gfCNCPoint1[19237] = {X 519.7998, Y 70.9591, Z -2.1667, A 0.000, B 0.000, C 0.000 }
gfCNCPoint1[19238] = {X 517.4110, Y 70.8403, Z -2.1667, A 0.000, B 0.000, C 0.000 }
gfCNCPoint1[19239] = {X 515.0458, Y 70.4852, Z -2.1667, A 0.000, B 0.000, C 0.000 }
gfCNCPoint1[19240] = {X 512.7275, Y 69.8971, Z -2.1667, A 0.000, B 0.000, C 0.000 }
gfCNCPoint1[19241] = {X 510.4789, Y 69.0820, Z -2.1667, A 0.000, B 0.000, C 0.000 }
gfCNCPoint1[19242] = {X 509.6264, Y 68.7046, Z -2.1667, A 0.000, B 0.000, C 0.000 }
gfCNCPoint1[19243] = {X 508.7892, Y 68.2944, Z -2.1667, A 0.000, B 0.000, C 0.000 }
gfCNCPoint1[19244] = {X 507.1705, Y 68.6592, Z -2.1667, A 0.000, B 0.000, C 0.000 }
gfCNCPoint1[19245] = {X 505.5305, Y 68.9117, Z -2.1667, A 0.000, B 0.000, C 0.000 }
gfCNCPoint1[19246] = {X 504.1120, Y 69.0379, Z -2.1667, A 0.000, B 0.000, C 0.000 }
gfCNCPoint1[19247] = {X 502.6885, Y 69.0800, Z -2.1667, A 0.000, B 0.000, C 0.000 }
gfCNCPoint1[19248] = {X 502.0391, Y 69.0800, Z -2.1667, A 0.000, B 0.000, C 0.000 }
gfCNCPoint1[19249] = {X 501.1772, Y 71.1329, Z -2.1667, A 0.000, B 0.000, C 0.000 }
gfCNCPoint1[19250] = {X 500.1596, Y 73.1132, Z -2.1667, A 0.000, B 0.000, C 0.000 }
gfCNCPoint1[19251] = {X 500.1596, Y 73.6949, Z -2.1667, A 0.000, B 0.000, C 0.000 }
gfCNCPoint1[19252] = {X 507.6819, Y 73.6949, Z -2.1667, A 0.000, B 0.000, C 0.000 }
gfCNCPoint1[19253] = {X 507.6819, Y 76.0949, Z -2.1667, A 0.000, B 0.000, C 0.000 }
gfCNCPoint1[19254] = {X 576.0965, Y 76.0949, Z -2.1667, A 0.000, B 0.000, C 0.000 }
gfCNCPoint1[19255] = {X 576.0965, Y 72.8901, Z -2.1667, A 0.000, B 0.000, C 0.000 }
gfCNCPoint1[19256] = {X 575.7178, Y 72.8147, Z -2.1667, A 0.000, B 0.000, C 0.000 }
gfCNCPoint1[19257] = {X 575.3401, Y 72.7341, Z -2.1667, A 0.000, B 0.000, C 0.000 }
gfCNCPoint1[19258] = {X 573.3201, Y 73.1034, Z -2.1667, A 0.000, B 0.000, C 0.000 }
gfCNCPoint1[19259] = {X 571.2786, Y 73.3258, Z -2.1667, A 0.000, B 0.000, C 0.000 }
gfCNCPoint1[19260] = {X 569.2264, Y 73.4000, Z -2.1667, A 0.000, B 0.000, C 0.000 }
gfCNCPoint1[19261] = {X 562.4443, Y 73.4000, Z -2.1667, A 0.000, B 0.000, C 0.000 }
gfCNCPoint1[19262] = {X 560.3341, Y 73.3215, Z -2.1667, A 0.000, B 0.000, C 0.000 }
gfCNCPoint1[19263] = {X 558.2355, Y 73.0864, Z -2.1667, A 0.000, B 0.000, C 0.000 }
gfCNCPoint1[19264] = {X 556.1603, Y 72.6960, Z -2.1667, A 0.000, B 0.000, C 0.000 }
gfCNCPoint1[19265] = {X 554.1197, Y 72.1526, Z -2.1667, A 0.000, B 0.000, C 0.000 }
gfCNCPoint1[19266] = {X 552.1252, Y 71.4590, Z -2.1667, A 0.000, B 0.000, C 0.000 }
gfCNCPoint1[19267] = {X 549.9757, Y 70.5165, Z -2.1667, A 0.000, B 0.000, C 0.000 }
gfCNCPoint1[19268] = {X 547.9113, Y 69.3999, Z -2.1667, A 0.000, B 0.000, C 0.000 }
gfCNCPoint1[19269] = {X 545.9462, Y 68.1165, Z -2.1667, A 0.000, B 0.000, C 0.000 }
gfCNCPoint1[19270] = {X 544.0938, Y 66.6753, Z -2.1667, A 0.000, B 0.000, C 0.000 }
gfCNCPoint1[19271] = {X 543.8496, Y 66.6765, Z -2.1667, A 0.000, B 0.000, C 0.000 }
gfCNCPoint1[19272] = {X 543.6054, Y 66.6749, Z -2.1667, A 0.000, B 0.000, C 0.000 }
gfCNCPoint1[19273] = {X 529.2683, Y 66.6753, Z -2.1667, A 0.000, B 0.000, C 0.000 }
gfCNCPoint1[19274] = {X 527.1808, Y 67.4783, Z -2.1667, A 0.000, B 0.000, C 0.000 }
gfCNCPoint1[19275] = {X 525.0223, Y 68.0636, Z -2.1667, A 0.000, B 0.000, C 0.000 }
gfCNCPoint1[19276] = {X 522.8151, Y 68.4251, Z -2.1667, A 0.000, B 0.000, C 0.000 }
gfCNCPoint1[19277] = {X 520.5826, Y 68.5589, Z -2.1667, A 0.000, B 0.000, C 0.000 }
gfCNCPoint1[19278] = {X 519.7998, Y 68.5591, Z -2.1667, A 0.000, B 0.000, C 0.000 }
gfCNCPoint1[19279] = {X 517.5593, Y 68.4430, Z -2.1667, A 0.000, B 0.000, C 0.000 }
gfCNCPoint1[19280] = {X 515.3429, Y 68.0961, Z -2.1667, A 0.000, B 0.000, C 0.000 }
gfCNCPoint1[19281] = {X 513.1742, Y 67.5219, Z -2.1667, A 0.000, B 0.000, C 0.000 }
gfCNCPoint1[19282] = {X 511.0764, Y 66.7267, Z -2.1667, A 0.000, B 0.000, C 0.000 }
gfCNCPoint1[19283] = {X 509.0720, Y 65.7189, Z -2.1667, A 0.000, B 0.000, C 0.000 }
gfCNCPoint1[19284] = {X 506.9797, Y 66.2511, Z -2.1667, A 0.000, B 0.000, C 0.000 }
gfCNCPoint1[19285] = {X 504.8448, Y 66.5725, Z -2.1667, A 0.000, B 0.000, C 0.000 }
gfCNCPoint1[19286] = {X 502.6885, Y 66.6800, Z -2.1667, A 0.000, B 0.000, C 0.000 }
gfCNCPoint1[19287] = {X 500.3217, Y 66.6800, Z -2.1667, A 0.000, B 0.000, C 0.000 }
gfCNCPoint1[19288] = {X 499.6229, Y 68.6759, Z -2.1667, A 0.000, B 0.000, C 0.000 }
gfCNCPoint1[19289] = {X 498.7670, Y 70.6096, Z -2.1667, A 0.000, B 0.000, C 0.000 }
gfCNCPoint1[19290] = {X 497.7596, Y 72.4689, Z -2.1667, A 0.000, B 0.000, C 0.000 }
gfCNCPoint1[19291] = {X 497.7596, Y 76.0949, Z -2.1667, A 0.000, B 0.000, C 0.000 }
gfCNCPoint1[19292] = {X 507.6819, Y 76.0949, Z -2.1667, A 0.000, B 0.000, C 0.000 }
gfCNCPoint1[19293] = {X 507.6819, Y 78.4949, Z -2.1667, A 0.000, B 0.000, C 0.000 }
gfCNCPoint1[19294] = {X 578.4965, Y 78.4949, Z -2.1667, A 0.000, B 0.000, C 0.000 }
gfCNCPoint1[19295] = {X 578.4965, Y 70.8313, Z -2.1667, A 0.000, B 0.000, C 0.000 }
gfCNCPoint1[19296] = {X 576.9097, Y 70.5998, Z -2.1667, A 0.000, B 0.000, C 0.000 }
gfCNCPoint1[19297] = {X 575.3401, Y 70.2710, Z -2.1667, A 0.000, B 0.000, C 0.000 }
gfCNCPoint1[19298] = {X 573.3236, Y 70.6751, Z -2.1667, A 0.000, B 0.000, C 0.000 }
gfCNCPoint1[19299] = {X 571.2815, Y 70.9187, Z -2.1667, A 0.000, B 0.000, C 0.000 }
gfCNCPoint1[19300] = {X 569.2264, Y 71.0000, Z -2.1667, A 0.000, B 0.000, C 0.000 }
gfCNCPoint1[19301] = {X 562.4443, Y 71.0000, Z -2.1667, A 0.000, B 0.000, C 0.000 }
gfCNCPoint1[19302] = {X 560.0511, Y 70.8896, Z -2.1667, A 0.000, B 0.000, C 0.000 }
gfCNCPoint1[19303] = {X 557.6782, Y 70.5594, Z -2.1667, A 0.000, B 0.000, C 0.000 }
gfCNCPoint1[19304] = {X 555.3457, Y 70.0122, Z -2.1667, A 0.000, B 0.000, C 0.000 }
gfCNCPoint1[19305] = {X 553.0736, Y 69.2526, Z -2.1667, A 0.000, B 0.000, C 0.000 }
gfCNCPoint1[19306] = {X 550.8810, Y 68.2871, Z -2.1667, A 0.000, B 0.000, C 0.000 }
gfCNCPoint1[19307] = {X 548.7866, Y 67.1239, Z -2.1667, A 0.000, B 0.000, C 0.000 }
gfCNCPoint1[19308] = {X 546.8081, Y 65.7728, Z -2.1667, A 0.000, B 0.000, C 0.000 }
gfCNCPoint1[19309] = {X 544.9624, Y 64.2454, Z -2.1667, A 0.000, B 0.000, C 0.000 }
gfCNCPoint1[19310] = {X 544.2916, Y 64.2718, Z -2.1667, A 0.000, B 0.000, C 0.000 }
gfCNCPoint1[19311] = {X 543.6203, Y 64.2749, Z -2.1667, A 0.000, B 0.000, C 0.000 }
gfCNCPoint1[19312] = {X 528.7431, Y 64.2753, Z -2.1667, A 0.000, B 0.000, C 0.000 }
gfCNCPoint1[19313] = {X 526.7893, Y 65.0775, Z -2.1667, A 0.000, B 0.000, C 0.000 }
gfCNCPoint1[19314] = {X 524.7600, Y 65.6630, Z -2.1667, A 0.000, B 0.000, C 0.000 }
gfCNCPoint1[19315] = {X 522.6791, Y 66.0249, Z -2.1667, A 0.000, B 0.000, C 0.000 }
gfCNCPoint1[19316] = {X 520.5713, Y 66.1589, Z -2.1667, A 0.000, B 0.000, C 0.000 }
gfCNCPoint1[19317] = {X 519.7998, Y 66.1591, Z -2.1667, A 0.000, B 0.000, C 0.000 }
gfCNCPoint1[19318] = {X 517.9641, Y 66.0715, Z -2.1667, A 0.000, B 0.000, C 0.000 }
gfCNCPoint1[19319] = {X 516.1450, Y 65.8096, Z -2.1667, A 0.000, B 0.000, C 0.000 }
gfCNCPoint1[19320] = {X 514.3592, Y 65.3756, Z -2.1667, A 0.000, B 0.000, C 0.000 }
gfCNCPoint1[19321] = {X 512.6228, Y 64.7735, Z -2.1667, A 0.000, B 0.000, C 0.000 }
gfCNCPoint1[19322] = {X 510.9516, Y 64.0089, Z -2.1667, A 0.000, B 0.000, C 0.000 }
gfCNCPoint1[19323] = {X 509.3609, Y 63.0886, Z -2.1667, A 0.000, B 0.000, C 0.000 }
gfCNCPoint1[19324] = {X 507.7389, Y 63.6068, Z -2.1667, A 0.000, B 0.000, C 0.000 }
gfCNCPoint1[19325] = {X 506.0774, Y 63.9798, Z -2.1667, A 0.000, B 0.000, C 0.000 }
gfCNCPoint1[19326] = {X 504.3896, Y 64.2048, Z -2.1667, A 0.000, B 0.000, C 0.000 }
gfCNCPoint1[19327] = {X 502.6885, Y 64.2800, Z -2.1667, A 0.000, B 0.000, C 0.000 }
gfCNCPoint1[19328] = {X 498.4791, Y 64.2800, Z -2.1667, A 0.000, B 0.000, C 0.000 }
gfCNCPoint1[19329] = {X 497.9415, Y 66.2507, Z -2.1667, A 0.000, B 0.000, C 0.000 }
gfCNCPoint1[19330] = {X 497.2388, Y 68.1688, Z -2.1667, A 0.000, B 0.000, C 0.000 }
gfCNCPoint1[19331] = {X 496.3761, Y 70.0204, Z -2.1667, A 0.000, B 0.000, C 0.000 }
gfCNCPoint1[19332] = {X 495.3596, Y 71.7923, Z -2.1667, A 0.000, B 0.000, C 0.000 }
gfCNCPoint1[19333] = {X 495.3597, Y 78.4949, Z -2.1667, A 0.000, B 0.000, C 0.000 }
gfCNCPoint1[19334] = {X 507.6819, Y 78.4949, Z -2.1667, A 0.000, B 0.000, C 0.000 }
gfCNCPoint1[19335] = {X 507.6819, Y 80.8949, Z -2.1667, A 0.000, B 0.000, C 0.000 }
gfCNCPoint1[19336] = {X 580.8965, Y 80.8949, Z -2.1667, A 0.000, B 0.000, C 0.000 }
gfCNCPoint1[19337] = {X 580.8965, Y 68.5934, Z -2.1667, A 0.000, B 0.000, C 0.000 }
gfCNCPoint1[19338] = {X 579.0251, Y 68.4747, Z -2.1667, A 0.000, B 0.000, C 0.000 }
gfCNCPoint1[19339] = {X 577.1691, Y 68.2078, Z -2.1667, A 0.000, B 0.000, C 0.000 }
gfCNCPoint1[19340] = {X 575.3401, Y 67.7943, Z -2.1667, A 0.000, B 0.000, C 0.000 }
gfCNCPoint1[19341] = {X 573.3283, Y 68.2408, Z -2.1667, A 0.000, B 0.000, C 0.000 }
gfCNCPoint1[19342] = {X 571.2852, Y 68.5100, Z -2.1667, A 0.000, B 0.000, C 0.000 }
gfCNCPoint1[19343] = {X 569.2264, Y 68.6000, Z -2.1667, A 0.000, B 0.000, C 0.000 }
gfCNCPoint1[19344] = {X 562.4443, Y 68.6000, Z -2.1667, A 0.000, B 0.000, C 0.000 }
gfCNCPoint1[19345] = {X 560.1442, Y 68.4876, Z -2.1667, A 0.000, B 0.000, C 0.000 }
gfCNCPoint1[19346] = {X 557.8659, Y 68.1516, Z -2.1667, A 0.000, B 0.000, C 0.000 }
gfCNCPoint1[19347] = {X 555.6313, Y 67.5952, Z -2.1667, A 0.000, B 0.000, C 0.000 }
gfCNCPoint1[19348] = {X 553.4615, Y 66.8236, Z -2.1667, A 0.000, B 0.000, C 0.000 }
gfCNCPoint1[19349] = {X 551.3773, Y 65.8442, Z -2.1667, A 0.000, B 0.000, C 0.000 }
gfCNCPoint1[19350] = {X 549.3984, Y 64.6664, Z -2.1667, A 0.000, B 0.000, C 0.000 }
gfCNCPoint1[19351] = {X 547.5438, Y 63.3012, Z -2.1667, A 0.000, B 0.000, C 0.000 }
gfCNCPoint1[19352] = {X 545.8311, Y 61.7619, Z -2.1667, A 0.000, B 0.000, C 0.000 }
gfCNCPoint1[19353] = {X 544.7354, Y 61.8541, Z -2.1667, A 0.000, B 0.000, C 0.000 }
gfCNCPoint1[19354] = {X 543.6361, Y 61.8749, Z -2.1667, A 0.000, B 0.000, C 0.000 }
gfCNCPoint1[19355] = {X 528.1826, Y 61.8754, Z -2.1667, A 0.000, B 0.000, C 0.000 }
gfCNCPoint1[19356] = {X 526.3697, Y 62.6774, Z -2.1667, A 0.000, B 0.000, C 0.000 }
gfCNCPoint1[19357] = {X 524.4760, Y 63.2635, Z -2.1667, A 0.000, B 0.000, C 0.000 }
gfCNCPoint1[19358] = {X 522.5270, Y 63.6257, Z -2.1667, A 0.000, B 0.000, C 0.000 }
gfCNCPoint1[19359] = {X 520.5492, Y 63.7590, Z -2.1667, A 0.000, B 0.000, C 0.000 }
gfCNCPoint1[19360] = {X 519.7998, Y 63.7591, Z -2.1667, A 0.000, B 0.000, C 0.000 }
gfCNCPoint1[19361] = {X 517.9902, Y 63.6618, Z -2.1667, A 0.000, B 0.000, C 0.000 }
gfCNCPoint1[19362] = {X 516.2015, Y 63.3711, Z -2.1667, A 0.000, B 0.000, C 0.000 }
gfCNCPoint1[19363] = {X 514.4543, Y 62.8904, Z -2.1667, A 0.000, B 0.000, C 0.000 }
gfCNCPoint1[19364] = {X 512.7687, Y 62.2251, Z -2.1667, A 0.000, B 0.000, C 0.000 }
gfCNCPoint1[19365] = {X 511.1641, Y 61.3829, Z -2.1667, A 0.000, B 0.000, C 0.000 }
gfCNCPoint1[19366] = {X 509.6590, Y 60.3735, Z -2.1667, A 0.000, B 0.000, C 0.000 }
gfCNCPoint1[19367] = {X 507.9866, Y 61.0270, Z -2.1667, A 0.000, B 0.000, C 0.000 }
gfCNCPoint1[19368] = {X 506.2542, Y 61.4991, Z -2.1667, A 0.000, B 0.000, C 0.000 }
gfCNCPoint1[19369] = {X 504.4815, Y 61.7845, Z -2.1667, A 0.000, B 0.000, C 0.000 }
gfCNCPoint1[19370] = {X 502.6885, Y 61.8800, Z -2.1667, A 0.000, B 0.000, C 0.000 }
gfCNCPoint1[19371] = {X 496.4789, Y 61.8800, Z -2.1667, A 0.000, B 0.000, C 0.000 }
gfCNCPoint1[19372] = {X 496.1191, Y 63.8335, Z -2.1667, A 0.000, B 0.000, C 0.000 }
gfCNCPoint1[19373] = {X 495.5821, Y 65.7458, Z -2.1667, A 0.000, B 0.000, C 0.000 }
gfCNCPoint1[19374] = {X 494.8723, Y 67.6009, Z -2.1667, A 0.000, B 0.000, C 0.000 }
gfCNCPoint1[19375] = {X 493.9957, Y 69.3833, Z -2.1667, A 0.000, B 0.000, C 0.000 }
gfCNCPoint1[19376] = {X 492.9596, Y 71.0780, Z -2.1667, A 0.000, B 0.000, C 0.000 }
gfCNCPoint1[19377] = {X 492.9597, Y 80.8949, Z -2.1667, A 0.000, B 0.000, C 0.000 }
gfCNCPoint1[19378] = {X 507.6819, Y 80.8949, Z -2.1667, A 0.000, B 0.000, C 0.000 }
gfCNCPoint1[19379] = {X 507.6819, Y 83.2949, Z -2.1667, A 0.000, B 0.000, C 0.000 }
gfCNCPoint1[19380] = {X 583.2965, Y 83.2949, Z -2.1667, A 0.000, B 0.000, C 0.000 }
gfCNCPoint1[19381] = {X 583.2965, Y 66.1198, Z -2.1667, A 0.000, B 0.000, C 0.000 }
gfCNCPoint1[19382] = {X 581.2871, Y 66.1993, Z -2.1667, A 0.000, B 0.000, C 0.000 }
gfCNCPoint1[19383] = {X 579.2793, Y 66.0882, Z -2.1667, A 0.000, B 0.000, C 0.000 }
gfCNCPoint1[19384] = {X 577.2910, Y 65.7873, Z -2.1667, A 0.000, B 0.000, C 0.000 }
gfCNCPoint1[19385] = {X 575.3401, Y 65.2993, Z -2.1667, A 0.000, B 0.000, C 0.000 }
gfCNCPoint1[19386] = {X 573.3348, Y 65.7981, Z -2.1667, A 0.000, B 0.000, C 0.000 }
gfCNCPoint1[19387] = {X 571.2904, Y 66.0993, Z -2.1667, A 0.000, B 0.000, C 0.000 }
gfCNCPoint1[19388] = {X 569.2264, Y 66.2000, Z -2.1667, A 0.000, B 0.000, C 0.000 }
gfCNCPoint1[19389] = {X 562.4443, Y 66.2000, Z -2.1667, A 0.000, B 0.000, C 0.000 }
gfCNCPoint1[19390] = {X 560.2302, Y 66.0841, Z -2.1667, A 0.000, B 0.000, C 0.000 }
gfCNCPoint1[19391] = {X 558.0403, Y 65.7375, Z -2.1667, A 0.000, B 0.000, C 0.000 }
gfCNCPoint1[19392] = {X 555.8985, Y 65.1641, Z -2.1667, A 0.000, B 0.000, C 0.000 }
gfCNCPoint1[19393] = {X 553.8284, Y 64.3702, Z -2.1667, A 0.000, B 0.000, C 0.000 }
gfCNCPoint1[19394] = {X 551.8525, Y 63.3644, Z -2.1667, A 0.000, B 0.000, C 0.000 }
gfCNCPoint1[19395] = {X 549.9924, Y 62.1578, Z -2.1667, A 0.000, B 0.000, C 0.000 }
gfCNCPoint1[19396] = {X 548.2685, Y 60.7635, Z -2.1667, A 0.000, B 0.000, C 0.000 }
gfCNCPoint1[19397] = {X 546.6997, Y 59.1968, Z -2.1667, A 0.000, B 0.000, C 0.000 }
gfCNCPoint1[19398] = {X 545.1838, Y 59.4165, Z -2.1667, A 0.000, B 0.000, C 0.000 }
gfCNCPoint1[19399] = {X 543.6531, Y 59.4749, Z -2.1667, A 0.000, B 0.000, C 0.000 }
gfCNCPoint1[19400] = {X 527.5785, Y 59.4754, Z -2.1667, A 0.000, B 0.000, C 0.000 }
gfCNCPoint1[19401] = {X 525.9214, Y 60.2760, Z -2.1667, A 0.000, B 0.000, C 0.000 }
gfCNCPoint1[19402] = {X 524.1770, Y 60.8624, Z -2.1667, A 0.000, B 0.000, C 0.000 }
gfCNCPoint1[19403] = {X 522.3727, Y 61.2253, Z -2.1667, A 0.000, B 0.000, C 0.000 }
gfCNCPoint1[19404] = {X 520.5372, Y 61.3590, Z -2.1667, A 0.000, B 0.000, C 0.000 }
gfCNCPoint1[19405] = {X 519.7998, Y 61.3591, Z -2.1667, A 0.000, B 0.000, C 0.000 }
gfCNCPoint1[19406] = {X 518.0043, Y 61.2474, Z -2.1667, A 0.000, B 0.000, C 0.000 }
gfCNCPoint1[19407] = {X 516.2365, Y 60.9138, Z -2.1667, A 0.000, B 0.000, C 0.000 }
gfCNCPoint1[19408] = {X 514.5237, Y 60.3637, Z -2.1667, A 0.000, B 0.000, C 0.000 }
gfCNCPoint1[19409] = {X 512.8923, Y 59.6054, Z -2.1667, A 0.000, B 0.000, C 0.000 }
gfCNCPoint1[19410] = {X 511.3676, Y 58.6507, Z -2.1667, A 0.000, B 0.000, C 0.000 }
gfCNCPoint1[19411] = {X 509.9730, Y 57.5142, Z -2.1667, A 0.000, B 0.000, C 0.000 }
gfCNCPoint1[19412] = {X 508.6156, Y 58.2113, Z -2.1667, A 0.000, B 0.000, C 0.000 }
gfCNCPoint1[19413] = {X 507.1924, Y 58.7617, Z -2.1667, A 0.000, B 0.000, C 0.000 }
gfCNCPoint1[19414] = {X 505.7192, Y 59.1593, Z -2.1667, A 0.000, B 0.000, C 0.000 }
gfCNCPoint1[19415] = {X 504.2123, Y 59.3996, Z -2.1667, A 0.000, B 0.000, C 0.000 }
gfCNCPoint1[19416] = {X 502.6885, Y 59.4800, Z -2.1667, A 0.000, B 0.000, C 0.000 }
gfCNCPoint1[19417] = {X 496.2450, Y 59.4800, Z -2.1667, A 0.000, B 0.000, C 0.000 }
gfCNCPoint1[19418] = {X 495.2580, Y 59.4463, Z -2.1667, A 0.000, B 0.000, C 0.000 }
gfCNCPoint1[19419] = {X 494.2756, Y 59.3454, Z -2.1667, A 0.000, B 0.000, C 0.000 }
gfCNCPoint1[19420] = {X 494.1342, Y 61.3007, Z -2.1667, A 0.000, B 0.000, C 0.000 }
gfCNCPoint1[19421] = {X 493.7949, Y 63.2316, Z -2.1667, A 0.000, B 0.000, C 0.000 }
gfCNCPoint1[19422] = {X 493.2614, Y 65.1180, Z -2.1667, A 0.000, B 0.000, C 0.000 }
gfCNCPoint1[19423] = {X 492.5390, Y 66.9405, Z -2.1667, A 0.000, B 0.000, C 0.000 }
gfCNCPoint1[19424] = {X 491.6353, Y 68.6801, Z -2.1667, A 0.000, B 0.000, C 0.000 }
gfCNCPoint1[19425] = {X 490.5596, Y 70.3191, Z -2.1667, A 0.000, B 0.000, C 0.000 }
gfCNCPoint1[19426] = {X 490.5597, Y 83.2949, Z -2.1667, A 0.000, B 0.000, C 0.000 }
gfCNCPoint1[19427] = {X 507.6819, Y 83.2949, Z -2.1667, A 0.000, B 0.000, C 0.000 }
gfCNCPoint1[19428] = {X 507.6819, Y 85.6949, Z -2.1667, A 0.000, B 0.000, C 0.000 }
gfCNCPoint1[19429] = {X 585.6965, Y 85.6949, Z -2.1667, A 0.000, B 0.000, C 0.000 }
gfCNCPoint1[19430] = {X 585.6965, Y 63.3150, Z -2.1667, A 0.000, B 0.000, C 0.000 }
gfCNCPoint1[19431] = {X 584.3995, Y 63.5678, Z -2.1667, A 0.000, B 0.000, C 0.000 }
gfCNCPoint1[19432] = {X 583.0879, Y 63.7289, Z -2.1667, A 0.000, B 0.000, C 0.000 }
gfCNCPoint1[19433] = {X 581.1242, Y 63.7971, Z -2.1667, A 0.000, B 0.000, C 0.000 }
gfCNCPoint1[19434] = {X 579.1641, Y 63.6600, Z -2.1667, A 0.000, B 0.000, C 0.000 }
gfCNCPoint1[19435] = {X 577.2291, Y 63.3191, Z -2.1667, A 0.000, B 0.000, C 0.000 }
gfCNCPoint1[19436] = {X 575.3401, Y 62.7781, Z -2.1667, A 0.000, B 0.000, C 0.000 }
gfCNCPoint1[19437] = {X 573.3441, Y 63.3435, Z -2.1667, A 0.000, B 0.000, C 0.000 }
gfCNCPoint1[19438] = {X 571.2979, Y 63.6855, Z -2.1667, A 0.000, B 0.000, C 0.000 }
gfCNCPoint1[19439] = {X 569.2264, Y 63.8000, Z -2.1667, A 0.000, B 0.000, C 0.000 }
gfCNCPoint1[19440] = {X 562.4443, Y 63.8000, Z -2.1667, A 0.000, B 0.000, C 0.000 }
gfCNCPoint1[19441] = {X 560.5407, Y 63.7034, Z -2.1667, A 0.000, B 0.000, C 0.000 }
gfCNCPoint1[19442] = {X 558.6566, Y 63.4145, Z -2.1667, A 0.000, B 0.000, C 0.000 }
gfCNCPoint1[19443] = {X 556.8115, Y 62.9363, Z -2.1667, A 0.000, B 0.000, C 0.000 }
gfCNCPoint1[19444] = {X 555.0242, Y 62.2737, Z -2.1667, A 0.000, B 0.000, C 0.000 }
gfCNCPoint1[19445] = {X 553.3133, Y 61.4336, Z -2.1667, A 0.000, B 0.000, C 0.000 }
gfCNCPoint1[19446] = {X 551.6962, Y 60.4246, Z -2.1667, A 0.000, B 0.000, C 0.000 }
gfCNCPoint1[19447] = {X 550.1896, Y 59.2570, Z -2.1667, A 0.000, B 0.000, C 0.000 }
gfCNCPoint1[19448] = {X 548.8089, Y 57.9428, Z -2.1667, A 0.000, B 0.000, C 0.000 }
gfCNCPoint1[19449] = {X 547.5685, Y 56.4956, Z -2.1667, A 0.000, B 0.000, C 0.000 }
gfCNCPoint1[19450] = {X 546.2932, Y 56.8304, Z -2.1667, A 0.000, B 0.000, C 0.000 }
gfCNCPoint1[19451] = {X 544.9891, Y 57.0243, Z -2.1667, A 0.000, B 0.000, C 0.000 }
gfCNCPoint1[19452] = {X 543.6716, Y 57.0749, Z -2.1667, A 0.000, B 0.000, C 0.000 }
gfCNCPoint1[19453] = {X 526.9187, Y 57.0754, Z -2.1667, A 0.000, B 0.000, C 0.000 }
gfCNCPoint1[19454] = {X 525.4309, Y 57.8752, Z -2.1667, A 0.000, B 0.000, C 0.000 }
gfCNCPoint1[19455] = {X 523.8471, Y 58.4624, Z -2.1667, A 0.000, B 0.000, C 0.000 }
gfCNCPoint1[19456] = {X 522.1975, Y 58.8261, Z -2.1667, A 0.000, B 0.000, C 0.000 }
gfCNCPoint1[19457] = {X 520.5136, Y 58.9591, Z -2.1667, A 0.000, B 0.000, C 0.000 }
gfCNCPoint1[19458] = {X 519.7998, Y 58.9591, Z -2.1667, A 0.000, B 0.000, C 0.000 }
gfCNCPoint1[19459] = {X 518.2467, Y 58.8589, Z -2.1667, A 0.000, B 0.000, C 0.000 }
gfCNCPoint1[19460] = {X 516.7195, Y 58.5598, Z -2.1667, A 0.000, B 0.000, C 0.000 }
gfCNCPoint1[19461] = {X 515.2433, Y 58.0668, Z -2.1667, A 0.000, B 0.000, C 0.000 }
gfCNCPoint1[19462] = {X 513.8428, Y 57.3882, Z -2.1667, A 0.000, B 0.000, C 0.000 }
gfCNCPoint1[19463] = {X 512.5411, Y 56.5351, Z -2.1667, A 0.000, B 0.000, C 0.000 }
gfCNCPoint1[19464] = {X 511.3600, Y 55.5218, Z -2.1667, A 0.000, B 0.000, C 0.000 }
gfCNCPoint1[19465] = {X 510.3189, Y 54.3650, Z -2.1667, A 0.000, B 0.000, C 0.000 }
gfCNCPoint1[19466] = {X 508.9711, Y 55.3177, Z -2.1667, A 0.000, B 0.000, C 0.000 }
gfCNCPoint1[19467] = {X 507.5060, Y 56.0778, Z -2.1667, A 0.000, B 0.000, C 0.000 }
gfCNCPoint1[19468] = {X 505.9510, Y 56.6311, Z -2.1667, A 0.000, B 0.000, C 0.000 }
gfCNCPoint1[19469] = {X 504.3351, Y 56.9672, Z -2.1667, A 0.000, B 0.000, C 0.000 }
gfCNCPoint1[19470] = {X 502.6885, Y 57.0800, Z -2.1667, A 0.000, B 0.000, C 0.000 }
gfCNCPoint1[19471] = {X 496.2450, Y 57.0800, Z -2.1667, A 0.000, B 0.000, C 0.000 }
gfCNCPoint1[19472] = {X 495.4216, Y 57.0519, Z -2.1667, A 0.000, B 0.000, C 0.000 }
gfCNCPoint1[19473] = {X 494.6020, Y 56.9677, Z -2.1667, A 0.000, B 0.000, C 0.000 }
gfCNCPoint1[19474] = {X 493.1719, Y 56.6826, Z -2.1667, A 0.000, B 0.000, C 0.000 }
gfCNCPoint1[19475] = {X 491.7866, Y 56.2272, Z -2.1667, A 0.000, B 0.000, C 0.000 }
gfCNCPoint1[19476] = {X 491.8566, Y 57.1124, Z -2.1667, A 0.000, B 0.000, C 0.000 }
gfCNCPoint1[19477] = {X 491.8800, Y 58.0000, Z -2.1667, A 0.000, B 0.000, C 0.000 }
gfCNCPoint1[19478] = {X 491.8794, Y 59.0735, Z -2.1667, A 0.000, B 0.000, C 0.000 }
gfCNCPoint1[19479] = {X 491.8781, Y 59.1839, Z -2.1667, A 0.000, B 0.000, C 0.000 }
gfCNCPoint1[19480] = {X 491.8762, Y 59.2942, Z -2.1667, A 0.000, B 0.000, C 0.000 }
gfCNCPoint1[19481] = {X 491.7363, Y 61.1320, Z -2.1667, A 0.000, B 0.000, C 0.000 }
gfCNCPoint1[19482] = {X 491.3969, Y 62.9435, Z -2.1667, A 0.000, B 0.000, C 0.000 }
gfCNCPoint1[19483] = {X 490.8621, Y 64.7072, Z -2.1667, A 0.000, B 0.000, C 0.000 }
gfCNCPoint1[19484] = {X 490.1381, Y 66.4022, Z -2.1667, A 0.000, B 0.000, C 0.000 }
gfCNCPoint1[19485] = {X 489.2337, Y 68.0080, Z -2.1667, A 0.000, B 0.000, C 0.000 }
gfCNCPoint1[19486] = {X 488.1596, Y 69.5057, Z -2.1667, A 0.000, B 0.000, C 0.000 }
gfCNCPoint1[19487] = {X 488.1598, Y 85.6949, Z -2.1667, A 0.000, B 0.000, C 0.000 }
gfCNCPoint1[19488] = {X 507.6819, Y 85.6949, Z -2.1667, A 0.000, B 0.000, C 0.000 }
gfCNCPoint1[19489] = {X 507.6819, Y 88.0949, Z -2.1667, A 0.000, B 0.000, C 0.000 }
gfCNCPoint1[19490] = {X 588.0965, Y 88.0949, Z -2.1667, A 0.000, B 0.000, C 0.000 }
gfCNCPoint1[19491] = {X 588.0965, Y 60.4644, Z -2.1667, A 0.000, B 0.000, C 0.000 }
gfCNCPoint1[19492] = {X 587.7998, Y 60.3564, Z -2.1667, A 0.000, B 0.000, C 0.000 }
gfCNCPoint1[19493] = {X 587.5052, Y 60.2427, Z -2.1667, A 0.000, B 0.000, C 0.000 }
gfCNCPoint1[19494] = {X 586.3438, Y 60.6540, Z -2.1667, A 0.000, B 0.000, C 0.000 }
gfCNCPoint1[19495] = {X 585.1549, Y 60.9769, Z -2.1667, A 0.000, B 0.000, C 0.000 }
gfCNCPoint1[19496] = {X 583.5152, Y 61.2699, Z -2.1667, A 0.000, B 0.000, C 0.000 }
gfCNCPoint1[19497] = {X 581.8543, Y 61.3951, Z -2.1667, A 0.000, B 0.000, C 0.000 }
gfCNCPoint1[19498] = {X 580.1892, Y 61.3512, Z -2.1667, A 0.000, B 0.000, C 0.000 }
gfCNCPoint1[19499] = {X 578.5372, Y 61.1386, Z -2.1667, A 0.000, B 0.000, C 0.000 }
gfCNCPoint1[19500] = {X 576.9153, Y 60.7595, Z -2.1667, A 0.000, B 0.000, C 0.000 }
gfCNCPoint1[19501] = {X 575.3401, Y 60.2178, Z -2.1667, A 0.000, B 0.000, C 0.000 }
gfCNCPoint1[19502] = {X 573.8611, Y 60.7315, Z -2.1667, A 0.000, B 0.000, C 0.000 }
gfCNCPoint1[19503] = {X 572.3399, Y 61.1017, Z -2.1667, A 0.000, B 0.000, C 0.000 }
gfCNCPoint1[19504] = {X 570.7903, Y 61.3253, Z -2.1667, A 0.000, B 0.000, C 0.000 }
gfCNCPoint1[19505] = {X 569.2264, Y 61.4000, Z -2.1667, A 0.000, B 0.000, C 0.000 }
gfCNCPoint1[19506] = {X 562.4443, Y 61.4000, Z -2.1667, A 0.000, B 0.000, C 0.000 }
gfCNCPoint1[19507] = {X 560.5827, Y 61.2940, Z -2.1667, A 0.000, B 0.000, C 0.000 }
gfCNCPoint1[19508] = {X 558.7453, Y 60.9774, Z -2.1667, A 0.000, B 0.000, C 0.000 }
gfCNCPoint1[19509] = {X 556.9556, Y 60.4543, Z -2.1667, A 0.000, B 0.000, C 0.000 }
gfCNCPoint1[19510] = {X 555.2369, Y 59.7313, Z -2.1667, A 0.000, B 0.000, C 0.000 }
gfCNCPoint1[19511] = {X 553.6113, Y 58.8180, Z -2.1667, A 0.000, B 0.000, C 0.000 }
gfCNCPoint1[19512] = {X 552.0999, Y 57.7261, Z -2.1667, A 0.000, B 0.000, C 0.000 }
gfCNCPoint1[19513] = {X 550.7222, Y 56.4697, Z -2.1667, A 0.000, B 0.000, C 0.000 }
gfCNCPoint1[19514] = {X 549.4961, Y 55.0650, Z -2.1667, A 0.000, B 0.000, C 0.000 }
gfCNCPoint1[19515] = {X 548.4373, Y 53.5302, Z -2.1667, A 0.000, B 0.000, C 0.000 }
gfCNCPoint1[19516] = {X 547.3156, Y 54.0416, Z -2.1667, A 0.000, B 0.000, C 0.000 }
gfCNCPoint1[19517] = {X 546.1380, Y 54.4064, Z -2.1667, A 0.000, B 0.000, C 0.000 }
gfCNCPoint1[19518] = {X 544.9235, Y 54.6187, Z -2.1667, A 0.000, B 0.000, C 0.000 }
gfCNCPoint1[19519] = {X 543.6920, Y 54.6749, Z -2.1667, A 0.000, B 0.000, C 0.000 }
gfCNCPoint1[19520] = {X 526.1842, Y 54.6754, Z -2.1667, A 0.000, B 0.000, C 0.000 }
gfCNCPoint1[19521] = {X 524.8903, Y 55.4721, Z -2.1667, A 0.000, B 0.000, C 0.000 }
gfCNCPoint1[19522] = {X 523.4892, Y 56.0601, Z -2.1667, A 0.000, B 0.000, C 0.000 }
gfCNCPoint1[19523] = {X 522.0142, Y 56.4254, Z -2.1667, A 0.000, B 0.000, C 0.000 }
gfCNCPoint1[19524] = {X 520.5006, Y 56.5591, Z -2.1667, A 0.000, B 0.000, C 0.000 }
gfCNCPoint1[19525] = {X 519.7998, Y 56.5591, Z -2.1667, A 0.000, B 0.000, C 0.000 }
gfCNCPoint1[19526] = {X 518.3493, Y 56.4498, Z -2.1667, A 0.000, B 0.000, C 0.000 }
gfCNCPoint1[19527] = {X 516.9316, Y 56.1244, Z -2.1667, A 0.000, B 0.000, C 0.000 }
gfCNCPoint1[19528] = {X 515.5787, Y 55.5903, Z -2.1667, A 0.000, B 0.000, C 0.000 }
gfCNCPoint1[19529] = {X 514.3210, Y 54.8595, Z -2.1667, A 0.000, B 0.000, C 0.000 }
gfCNCPoint1[19530] = {X 513.1871, Y 53.9484, Z -2.1667, A 0.000, B 0.000, C 0.000 }
gfCNCPoint1[19531] = {X 512.2025, Y 52.8778, Z -2.1667, A 0.000, B 0.000, C 0.000 }
gfCNCPoint1[19532] = {X 511.3855, Y 51.6648, Z -2.1667, A 0.000, B 0.000, C 0.000 }
gfCNCPoint1[19533] = {X 510.7606, Y 50.3426, Z -2.1667, A 0.000, B 0.000, C 0.000 }
gfCNCPoint1[19534] = {X 509.8636, Y 51.4977, Z -2.1667, A 0.000, B 0.000, C 0.000 }
gfCNCPoint1[19535] = {X 508.8029, Y 52.5044, Z -2.1667, A 0.000, B 0.000, C 0.000 }
gfCNCPoint1[19536] = {X 507.7229, Y 53.2678, Z -2.1667, A 0.000, B 0.000, C 0.000 }
gfCNCPoint1[19537] = {X 506.5489, Y 53.8769, Z -2.1667, A 0.000, B 0.000, C 0.000 }
gfCNCPoint1[19538] = {X 505.3028, Y 54.3203, Z -2.1667, A 0.000, B 0.000, C 0.000 }
gfCNCPoint1[19539] = {X 504.0080, Y 54.5896, Z -2.1667, A 0.000, B 0.000, C 0.000 }
gfCNCPoint1[19540] = {X 502.6885, Y 54.6800, Z -2.1667, A 0.000, B 0.000, C 0.000 }
gfCNCPoint1[19541] = {X 496.2450, Y 54.6800, Z -2.1667, A 0.000, B 0.000, C 0.000 }
gfCNCPoint1[19542] = {X 495.0285, Y 54.6033, Z -2.1667, A 0.000, B 0.000, C 0.000 }
gfCNCPoint1[19543] = {X 493.8313, Y 54.3742, Z -2.1667, A 0.000, B 0.000, C 0.000 }
gfCNCPoint1[19544] = {X 492.6724, Y 53.9966, Z -2.1667, A 0.000, B 0.000, C 0.000 }
gfCNCPoint1[19545] = {X 491.4451, Y 53.4062, Z -2.1667, A 0.000, B 0.000, C 0.000 }
gfCNCPoint1[19546] = {X 490.3129, Y 52.6493, Z -2.1667, A 0.000, B 0.000, C 0.000 }
gfCNCPoint1[19547] = {X 489.2980, Y 51.7410, Z -2.1667, A 0.000, B 0.000, C 0.000 }
gfCNCPoint1[19548] = {X 488.8683, Y 52.1573, Z -2.1667, A 0.000, B 0.000, C 0.000 }
gfCNCPoint1[19549] = {X 488.4137, Y 52.5463, Z -2.1667, A 0.000, B 0.000, C 0.000 }
gfCNCPoint1[19550] = {X 488.8649, Y 53.8245, Z -2.1667, A 0.000, B 0.000, C 0.000 }
gfCNCPoint1[19551] = {X 489.1946, Y 55.1393, Z -2.1667, A 0.000, B 0.000, C 0.000 }
gfCNCPoint1[19552] = {X 489.3999, Y 56.4792, Z -2.1667, A 0.000, B 0.000, C 0.000 }
gfCNCPoint1[19553] = {X 489.4600, Y 57.2386, Z -2.1667, A 0.000, B 0.000, C 0.000 }
gfCNCPoint1[19554] = {X 489.4800, Y 58.0000, Z -2.1667, A 0.000, B 0.000, C 0.000 }
gfCNCPoint1[19555] = {X 489.4795, Y 59.0537, Z -2.1667, A 0.000, B 0.000, C 0.000 }
gfCNCPoint1[19556] = {X 489.3595, Y 60.7979, Z -2.1667, A 0.000, B 0.000, C 0.000 }
gfCNCPoint1[19557] = {X 489.0302, Y 62.5150, Z -2.1667, A 0.000, B 0.000, C 0.000 }
gfCNCPoint1[19558] = {X 488.4964, Y 64.1799, Z -2.1667, A 0.000, B 0.000, C 0.000 }
gfCNCPoint1[19559] = {X 487.7657, Y 65.7682, Z -2.1667, A 0.000, B 0.000, C 0.000 }
gfCNCPoint1[19560] = {X 486.8490, Y 67.2570, Z -2.1667, A 0.000, B 0.000, C 0.000 }
gfCNCPoint1[19561] = {X 485.7595, Y 68.6244, Z -2.1667, A 0.000, B 0.000, C 0.000 }
gfCNCPoint1[19562] = {X 485.7598, Y 87.3800, Z -2.1667, A 0.000, B 0.000, C 0.000 }
gfCNCPoint1[19563] = {X 486.0676, Y 87.7326, Z -2.1667, A 0.000, B 0.000, C 0.000 }
gfCNCPoint1[19564] = {X 486.3638, Y 88.0949, Z -2.1667, A 0.000, B 0.000, C 0.000 }
gfCNCPoint1[19565] = {X 507.6819, Y 88.0949, Z -2.1667, A 0.000, B 0.000, C 0.000 }
gfCNCPoint1[19566] = {X 507.6819, Y 90.4949, Z -2.1667, A 0.000, B 0.000, C 0.000 }
gfCNCPoint1[19567] = {X 590.4965, Y 90.4949, Z -2.1667, A 0.000, B 0.000, C 0.000 }
gfCNCPoint1[19568] = {X 590.4965, Y 58.6615, Z -2.1667, A 0.000, B 0.000, C 0.000 }
gfCNCPoint1[19569] = {X 588.9714, Y 58.2279, Z -2.1667, A 0.000, B 0.000, C 0.000 }
gfCNCPoint1[19570] = {X 587.5052, Y 57.6246, Z -2.1667, A 0.000, B 0.000, C 0.000 }
gfCNCPoint1[19571] = {X 585.8387, Y 58.2956, Z -2.1667, A 0.000, B 0.000, C 0.000 }
gfCNCPoint1[19572] = {X 584.0999, Y 58.7477, Z -2.1667, A 0.000, B 0.000, C 0.000 }
gfCNCPoint1[19573] = {X 582.3176, Y 58.9733, Z -2.1667, A 0.000, B 0.000, C 0.000 }
gfCNCPoint1[19574] = {X 580.5210, Y 58.9689, Z -2.1667, A 0.000, B 0.000, C 0.000 }
gfCNCPoint1[19575] = {X 578.7398, Y 58.7344, Z -2.1667, A 0.000, B 0.000, C 0.000 }
gfCNCPoint1[19576] = {X 577.0034, Y 58.2738, Z -2.1667, A 0.000, B 0.000, C 0.000 }
gfCNCPoint1[19577] = {X 575.3401, Y 57.5945, Z -2.1667, A 0.000, B 0.000, C 0.000 }
gfCNCPoint1[19578] = {X 573.8813, Y 58.2035, Z -2.1667, A 0.000, B 0.000, C 0.000 }
gfCNCPoint1[19579] = {X 572.3630, Y 58.6441, Z -2.1667, A 0.000, B 0.000, C 0.000 }
gfCNCPoint1[19580] = {X 570.8048, Y 58.9107, Z -2.1667, A 0.000, B 0.000, C 0.000 }
gfCNCPoint1[19581] = {X 569.2264, Y 59.0000, Z -2.1667, A 0.000, B 0.000, C 0.000 }
gfCNCPoint1[19582] = {X 562.4443, Y 59.0000, Z -2.1667, A 0.000, B 0.000, C 0.000 }
gfCNCPoint1[19583] = {X 560.6576, Y 58.8855, Z -2.1667, A 0.000, B 0.000, C 0.000 }
gfCNCPoint1[19584] = {X 558.9000, Y 58.5439, Z -2.1667, A 0.000, B 0.000, C 0.000 }
gfCNCPoint1[19585] = {X 557.2005, Y 57.9808, Z -2.1667, A 0.000, B 0.000, C 0.000 }
gfCNCPoint1[19586] = {X 555.5867, Y 57.2054, Z -2.1667, A 0.000, B 0.000, C 0.000 }
gfCNCPoint1[19587] = {X 554.0850, Y 56.2304, Z -2.1667, A 0.000, B 0.000, C 0.000 }
gfCNCPoint1[19588] = {X 552.7201, Y 55.0717, Z -2.1667, A 0.000, B 0.000, C 0.000 }
gfCNCPoint1[19589] = {X 551.5142, Y 53.7483, Z -2.1667, A 0.000, B 0.000, C 0.000 }
gfCNCPoint1[19590] = {X 550.4871, Y 52.2818, Z -2.1667, A 0.000, B 0.000, C 0.000 }
gfCNCPoint1[19591] = {X 549.8374, Y 51.0881, Z -2.1667, A 0.000, B 0.000, C 0.000 }
gfCNCPoint1[19592] = {X 549.3065, Y 49.8371, Z -2.1667, A 0.000, B 0.000, C 0.000 }
gfCNCPoint1[19593] = {X 548.3751, Y 50.7139, Z -2.1667, A 0.000, B 0.000, C 0.000 }
gfCNCPoint1[19594] = {X 547.3047, Y 51.4142, Z -2.1667, A 0.000, B 0.000, C 0.000 }
gfCNCPoint1[19595] = {X 546.1632, Y 51.9051, Z -2.1667, A 0.000, B 0.000, C 0.000 }
gfCNCPoint1[19596] = {X 544.9550, Y 52.1948, Z -2.1667, A 0.000, B 0.000, C 0.000 }
gfCNCPoint1[19597] = {X 543.7152, Y 52.2749, Z -2.1667, A 0.000, B 0.000, C 0.000 }
gfCNCPoint1[19598] = {X 525.3420, Y 52.2754, Z -2.1667, A 0.000, B 0.000, C 0.000 }
gfCNCPoint1[19599] = {X 524.2749, Y 53.0670, Z -2.1667, A 0.000, B 0.000, C 0.000 }
gfCNCPoint1[19600] = {X 523.0841, Y 53.6562, Z -2.1667, A 0.000, B 0.000, C 0.000 }
gfCNCPoint1[19601] = {X 521.8075, Y 54.0241, Z -2.1667, A 0.000, B 0.000, C 0.000 }
gfCNCPoint1[19602] = {X 520.4857, Y 54.1591, Z -2.1667, A 0.000, B 0.000, C 0.000 }
gfCNCPoint1[19603] = {X 519.7998, Y 54.1591, Z -2.1667, A 0.000, B 0.000, C 0.000 }
gfCNCPoint1[19604] = {X 518.5529, Y 54.0515, Z -2.1667, A 0.000, B 0.000, C 0.000 }
gfCNCPoint1[19605] = {X 517.3428, Y 53.7320, Z -2.1667, A 0.000, B 0.000, C 0.000 }
gfCNCPoint1[19606] = {X 516.2054, Y 53.2099, Z -2.1667, A 0.000, B 0.000, C 0.000 }
gfCNCPoint1[19607] = {X 515.1742, Y 52.5007, Z -2.1667, A 0.000, B 0.000, C 0.000 }
gfCNCPoint1[19608] = {X 514.2797, Y 51.6254, Z -2.1667, A 0.000, B 0.000, C 0.000 }
gfCNCPoint1[19609] = {X 513.5483, Y 50.6098, Z -2.1667, A 0.000, B 0.000, C 0.000 }
gfCNCPoint1[19610] = {X 513.0017, Y 49.4839, Z -2.1667, A 0.000, B 0.000, C 0.000 }
gfCNCPoint1[19611] = {X 512.7353, Y 48.6374, Z -2.1667, A 0.000, B 0.000, C 0.000 }
gfCNCPoint1[19612] = {X 512.5739, Y 47.7649, Z -2.1667, A 0.000, B 0.000, C 0.000 }
gfCNCPoint1[19613] = {X 512.5198, Y 46.8791, Z -2.1667, A 0.000, B 0.000, C 0.000 }
gfCNCPoint1[19614] = {X 512.5198, Y 39.9011, Z -2.1667, A 0.000, B 0.000, C 0.000 }
gfCNCPoint1[19615] = {X 512.5807, Y 38.9616, Z -2.1667, A 0.000, B 0.000, C 0.000 }
gfCNCPoint1[19616] = {X 512.7623, Y 38.0378, Z -2.1667, A 0.000, B 0.000, C 0.000 }
gfCNCPoint1[19617] = {X 513.0616, Y 37.1451, Z -2.1667, A 0.000, B 0.000, C 0.000 }
gfCNCPoint1[19618] = {X 513.5571, Y 36.1558, Z -2.1667, A 0.000, B 0.000, C 0.000 }
gfCNCPoint1[19619] = {X 514.1968, Y 35.2530, Z -2.1667, A 0.000, B 0.000, C 0.000 }
gfCNCPoint1[19620] = {X 514.9659, Y 34.4576, Z -2.1667, A 0.000, B 0.000, C 0.000 }
gfCNCPoint1[19621] = {X 515.8467, Y 33.7879, Z -2.1667, A 0.000, B 0.000, C 0.000 }
gfCNCPoint1[19622] = {X 513.2402, Y 29.7572, Z -2.1667, A 0.000, B 0.000, C 0.000 }
gfCNCPoint1[19623] = {X 513.5213, Y 29.5809, Z -2.1667, A 0.000, B 0.000, C 0.000 }
gfCNCPoint1[19624] = {X 513.8071, Y 29.4123, Z -2.1667, A 0.000, B 0.000, C 0.000 }
gfCNCPoint1[19625] = {X 513.8074, Y 27.6761, Z -2.1667, A 0.000, B 0.000, C 0.000 }
gfCNCPoint1[19626] = {X 513.5214, Y 27.5010, Z -2.1667, A 0.000, B 0.000, C 0.000 }
gfCNCPoint1[19627] = {X 513.2403, Y 27.3181, Z -2.1667, A 0.000, B 0.000, C 0.000 }
gfCNCPoint1[19628] = {X 513.2402, Y 29.7572, Z -2.1667, A 0.000, B 0.000, C 0.000 }
gfCNCPoint1[19629] = {X 514.5435, Y 31.7725, Z -2.1667, A 0.000, B 0.000, C 0.000 }
gfCNCPoint1[19630] = {X 515.3543, Y 31.3022, Z -2.1667, A 0.000, B 0.000, C 0.000 }
gfCNCPoint1[19631] = {X 516.2069, Y 30.9126, Z -2.1667, A 0.000, B 0.000, C 0.000 }
gfCNCPoint1[19632] = {X 516.2077, Y 26.2050, Z -2.1667, A 0.000, B 0.000, C 0.000 }
gfCNCPoint1[19633] = {X 515.3713, Y 25.8041, Z -2.1667, A 0.000, B 0.000, C 0.000 }
gfCNCPoint1[19634] = {X 514.5771, Y 25.3249, Z -2.1667, A 0.000, B 0.000, C 0.000 }
gfCNCPoint1[19635] = {X 513.5937, Y 24.5697, Z -2.1667, A 0.000, B 0.000, C 0.000 }
gfCNCPoint1[19636] = {X 512.7148, Y 23.6949, Z -2.1667, A 0.000, B 0.000, C 0.000 }
gfCNCPoint1[19637] = {X 511.9551, Y 22.7150, Z -2.1667, A 0.000, B 0.000, C 0.000 }
gfCNCPoint1[19638] = {X 511.3268, Y 21.6460, Z -2.1667, A 0.000, B 0.000, C 0.000 }
gfCNCPoint1[19639] = {X 510.8403, Y 20.5055, Z -2.1667, A 0.000, B 0.000, C 0.000 }
gfCNCPoint1[19640] = {X 510.8402, Y 36.2365, Z -2.1667, A 0.000, B 0.000, C 0.000 }
gfCNCPoint1[19641] = {X 511.4991, Y 34.9211, Z -2.1667, A 0.000, B 0.000, C 0.000 }
gfCNCPoint1[19642] = {X 512.3496, Y 33.7207, Z -2.1667, A 0.000, B 0.000, C 0.000 }
gfCNCPoint1[19643] = {X 513.3723, Y 32.6630, Z -2.1667, A 0.000, B 0.000, C 0.000 }
gfCNCPoint1[19644] = {X 514.5435, Y 31.7725, Z -2.1667, A 0.000, B 0.000, C 0.000 }
gfCNCPoint1[19645] = {X 515.8467, Y 33.7879, Z -2.1667, A 0.000, B 0.000, C 0.000 }
gfCNCPoint1[19646] = {X 516.7433, Y 33.2938, Z -2.1667, A 0.000, B 0.000, C 0.000 }
gfCNCPoint1[19647] = {X 517.7004, Y 32.9304, Z -2.1667, A 0.000, B 0.000, C 0.000 }
gfCNCPoint1[19648] = {X 518.6990, Y 32.7048, Z -2.1667, A 0.000, B 0.000, C 0.000 }
gfCNCPoint1[19649] = {X 518.6299, Y 32.1290, Z -2.1667, A 0.000, B 0.000, C 0.000 }
gfCNCPoint1[19650] = {X 518.6068, Y 31.5495, Z -2.1667, A 0.000, B 0.000, C 0.000 }
gfCNCPoint1[19651] = {X 518.6080, Y 24.4373, Z -2.1667, A 0.000, B 0.000, C 0.000 }
gfCNCPoint1[19652] = {X 517.3908, Y 24.0939, Z -2.1667, A 0.000, B 0.000, C 0.000 }
gfCNCPoint1[19653] = {X 516.2515, Y 23.5449, Z -2.1667, A 0.000, B 0.000, C 0.000 }
gfCNCPoint1[19654] = {X 515.2243, Y 22.8071, Z -2.1667, A 0.000, B 0.000, C 0.000 }
gfCNCPoint1[19655] = {X 514.3404, Y 21.9026, Z -2.1667, A 0.000, B 0.000, C 0.000 }
gfCNCPoint1[19656] = {X 513.6263, Y 20.8588, Z -2.1667, A 0.000, B 0.000, C 0.000 }
gfCNCPoint1[19657] = {X 513.1036, Y 19.7072, Z -2.1667, A 0.000, B 0.000, C 0.000 }
gfCNCPoint1[19658] = {X 512.7935, Y 18.5141, Z -2.1667, A 0.000, B 0.000, C 0.000 }
gfCNCPoint1[19659] = {X 512.6891, Y 17.2857, Z -2.1667, A 0.000, B 0.000, C 0.000 }
gfCNCPoint1[19660] = {X 512.6891, Y 10.3077, Z -2.1667, A 0.000, B 0.000, C 0.000 }
gfCNCPoint1[19661] = {X 512.7002, Y 9.9058, Z -2.1667, A 0.000, B 0.000, C 0.000 }
gfCNCPoint1[19662] = {X 512.7335, Y 9.5051, Z -2.1667, A 0.000, B 0.000, C 0.000 }
gfCNCPoint1[19663] = {X 509.4580, Y 9.5051, Z -2.1667, A 0.000, B 0.000, C 0.000 }
gfCNCPoint1[19664] = {X 509.7401, Y 10.3730, Z -2.1667, A 0.000, B 0.000, C 0.000 }
gfCNCPoint1[19665] = {X 509.9112, Y 11.2695, Z -2.1667, A 0.000, B 0.000, C 0.000 }
gfCNCPoint1[19666] = {X 509.9685, Y 12.1804, Z -2.1667, A 0.000, B 0.000, C 0.000 }
gfCNCPoint1[19667] = {X 509.9682, Y 13.0462, Z -2.1667, A 0.000, B 0.000, C 0.000 }
gfCNCPoint1[19668] = {X 509.8611, Y 14.2239, Z -2.1667, A 0.000, B 0.000, C 0.000 }
gfCNCPoint1[19669] = {X 509.5647, Y 15.3688, Z -2.1667, A 0.000, B 0.000, C 0.000 }
gfCNCPoint1[19670] = {X 509.0869, Y 16.4505, Z -2.1667, A 0.000, B 0.000, C 0.000 }
gfCNCPoint1[19671] = {X 508.4403, Y 17.4407, Z -2.1667, A 0.000, B 0.000, C 0.000 }
gfCNCPoint1[19672] = {X 508.4402, Y 39.7461, Z -2.1667, A 0.000, B 0.000, C 0.000 }
gfCNCPoint1[19673] = {X 509.0887, Y 40.7395, Z -2.1667, A 0.000, B 0.000, C 0.000 }
gfCNCPoint1[19674] = {X 509.5672, Y 41.8251, Z -2.1667, A 0.000, B 0.000, C 0.000 }
gfCNCPoint1[19675] = {X 509.8630, Y 42.9741, Z -2.1667, A 0.000, B 0.000, C 0.000 }
gfCNCPoint1[19676] = {X 509.9683, Y 44.1558, Z -2.1667, A 0.000, B 0.000, C 0.000 }
gfCNCPoint1[19677] = {X 509.9685, Y 45.0000, Z -2.1667, A 0.000, B 0.000, C 0.000 }
gfCNCPoint1[19678] = {X 509.8909, Y 46.0603, Z -2.1667, A 0.000, B 0.000, C 0.000 }
gfCNCPoint1[19679] = {X 509.6596, Y 47.0980, Z -2.1667, A 0.000, B 0.000, C 0.000 }
gfCNCPoint1[19680] = {X 509.2797, Y 48.0910, Z -2.1667, A 0.000, B 0.000, C 0.000 }
gfCNCPoint1[19681] = {X 508.7593, Y 49.0180, Z -2.1667, A 0.000, B 0.000, C 0.000 }
gfCNCPoint1[19682] = {X 508.0200, Y 49.9571, Z -2.1667, A 0.000, B 0.000, C 0.000 }
gfCNCPoint1[19683] = {X 507.1371, Y 50.7626, Z -2.1667, A 0.000, B 0.000, C 0.000 }
gfCNCPoint1[19684] = {X 506.1343, Y 51.4129, Z -2.1667, A 0.000, B 0.000, C 0.000 }
gfCNCPoint1[19685] = {X 505.0386, Y 51.8902, Z -2.1667, A 0.000, B 0.000, C 0.000 }
gfCNCPoint1[19686] = {X 503.8796, Y 52.1819, Z -2.1667, A 0.000, B 0.000, C 0.000 }
gfCNCPoint1[19687] = {X 502.6885, Y 52.2800, Z -2.1667, A 0.000, B 0.000, C 0.000 }
gfCNCPoint1[19688] = {X 496.2450, Y 52.2800, Z -2.1667, A 0.000, B 0.000, C 0.000 }
gfCNCPoint1[19689] = {X 495.0845, Y 52.1869, Z -2.1667, A 0.000, B 0.000, C 0.000 }
gfCNCPoint1[19690] = {X 493.9538, Y 51.9100, Z -2.1667, A 0.000, B 0.000, C 0.000 }
gfCNCPoint1[19691] = {X 492.8816, Y 51.4564, Z -2.1667, A 0.000, B 0.000, C 0.000 }
gfCNCPoint1[19692] = {X 491.8954, Y 50.8377, Z -2.1667, A 0.000, B 0.000, C 0.000 }
gfCNCPoint1[19693] = {X 491.0204, Y 50.0697, Z -2.1667, A 0.000, B 0.000, C 0.000 }
gfCNCPoint1[19694] = {X 490.2980, Y 49.1989, Z -2.1667, A 0.000, B 0.000, C 0.000 }
gfCNCPoint1[19695] = {X 489.7192, Y 48.2267, Z -2.1667, A 0.000, B 0.000, C 0.000 }
gfCNCPoint1[19696] = {X 489.2980, Y 47.1766, Z -2.1667, A 0.000, B 0.000, C 0.000 }
gfCNCPoint1[19697] = {X 488.8769, Y 48.2267, Z -2.1667, A 0.000, B 0.000, C 0.000 }
gfCNCPoint1[19698] = {X 488.2981, Y 49.1989, Z -2.1667, A 0.000, B 0.000, C 0.000 }
gfCNCPoint1[19699] = {X 487.5756, Y 50.0697, Z -2.1667, A 0.000, B 0.000, C 0.000 }
gfCNCPoint1[19700] = {X 486.8824, Y 50.6978, Z -2.1667, A 0.000, B 0.000, C 0.000 }
gfCNCPoint1[19701] = {X 486.1145, Y 51.2318, Z -2.1667, A 0.000, B 0.000, C 0.000 }
gfCNCPoint1[19702] = {X 485.2843, Y 51.6629, Z -2.1667, A 0.000, B 0.000, C 0.000 }
gfCNCPoint1[19703] = {X 486.0586, Y 53.1385, Z -2.1667, A 0.000, B 0.000, C 0.000 }
gfCNCPoint1[19704] = {X 486.6224, Y 54.7067, Z -2.1667, A 0.000, B 0.000, C 0.000 }
gfCNCPoint1[19705] = {X 486.9651, Y 56.3375, Z -2.1667, A 0.000, B 0.000, C 0.000 }
gfCNCPoint1[19706] = {X 487.0800, Y 58.0000, Z -2.1667, A 0.000, B 0.000, C 0.000 }
gfCNCPoint1[19707] = {X 487.0796, Y 59.0339, Z -2.1667, A 0.000, B 0.000, C 0.000 }
gfCNCPoint1[19708] = {X 486.9596, Y 60.6354, Z -2.1667, A 0.000, B 0.000, C 0.000 }
gfCNCPoint1[19709] = {X 486.6282, Y 62.2068, Z -2.1667, A 0.000, B 0.000, C 0.000 }
gfCNCPoint1[19710] = {X 486.0913, Y 63.7204, Z -2.1667, A 0.000, B 0.000, C 0.000 }
gfCNCPoint1[19711] = {X 485.3584, Y 65.1493, Z -2.1667, A 0.000, B 0.000, C 0.000 }
gfCNCPoint1[19712] = {X 484.4424, Y 66.4685, Z -2.1667, A 0.000, B 0.000, C 0.000 }
gfCNCPoint1[19713] = {X 483.3595, Y 67.6544, Z -2.1667, A 0.000, B 0.000, C 0.000 }
gfCNCPoint1[19714] = {X 483.3598, Y 88.3511, Z -2.1667, A 0.000, B 0.000, C 0.000 }
gfCNCPoint1[19715] = {X 484.3097, Y 89.3716, Z -2.1667, A 0.000, B 0.000, C 0.000 }
gfCNCPoint1[19716] = {X 485.1353, Y 90.4949, Z -2.1667, A 0.000, B 0.000, C 0.000 }
gfCNCPoint1[19717] = {X 507.6819, Y 90.4949, Z -2.1667, A 0.000, B 0.000, C 0.000 }
gfCNCPoint1[19718] = {X 507.6819, Y 92.8949, Z -2.1667, A 0.000, B 0.000, C 0.000 }
gfCNCPoint1[19719] = {X 592.8965, Y 92.8949, Z -2.1667, A 0.000, B 0.000, C 0.000 }
gfCNCPoint1[19720] = {X 592.8965, Y 56.5812, Z -2.1667, A 0.000, B 0.000, C 0.000 }
gfCNCPoint1[19721] = {X 591.4809, Y 56.4128, Z -2.1667, A 0.000, B 0.000, C 0.000 }
gfCNCPoint1[19722] = {X 590.0967, Y 56.0720, Z -2.1667, A 0.000, B 0.000, C 0.000 }
gfCNCPoint1[19723] = {X 588.7648, Y 55.5640, Z -2.1667, A 0.000, B 0.000, C 0.000 }
gfCNCPoint1[19724] = {X 587.5052, Y 54.8965, Z -2.1667, A 0.000, B 0.000, C 0.000 }
gfCNCPoint1[19725] = {X 586.9690, Y 55.2051, Z -2.1667, A 0.000, B 0.000, C 0.000 }
gfCNCPoint1[19726] = {X 586.4171, Y 55.4846, Z -2.1667, A 0.000, B 0.000, C 0.000 }
gfCNCPoint1[19727] = {X 584.8782, Y 56.0830, Z -2.1667, A 0.000, B 0.000, C 0.000 }
gfCNCPoint1[19728] = {X 583.2699, Y 56.4570, Z -2.1667, A 0.000, B 0.000, C 0.000 }
gfCNCPoint1[19729] = {X 581.6248, Y 56.5987, Z -2.1667, A 0.000, B 0.000, C 0.000 }
gfCNCPoint1[19730] = {X 579.9763, Y 56.5055, Z -2.1667, A 0.000, B 0.000, C 0.000 }
gfCNCPoint1[19731] = {X 578.3577, Y 56.1792, Z -2.1667, A 0.000, B 0.000, C 0.000 }
gfCNCPoint1[19732] = {X 576.8018, Y 55.6263, Z -2.1667, A 0.000, B 0.000, C 0.000 }
gfCNCPoint1[19733] = {X 575.3401, Y 54.8581, Z -2.1667, A 0.000, B 0.000, C 0.000 }
gfCNCPoint1[19734] = {X 573.9176, Y 55.6091, Z -2.1667, A 0.000, B 0.000, C 0.000 }
gfCNCPoint1[19735] = {X 572.4049, Y 56.1560, Z -2.1667, A 0.000, B 0.000, C 0.000 }
gfCNCPoint1[19736] = {X 570.8311, Y 56.4885, Z -2.1667, A 0.000, B 0.000, C 0.000 }
gfCNCPoint1[19737] = {X 569.2264, Y 56.6000, Z -2.1667, A 0.000, B 0.000, C 0.000 }
gfCNCPoint1[19738] = {X 562.4443, Y 56.6000, Z -2.1667, A 0.000, B 0.000, C 0.000 }
gfCNCPoint1[19739] = {X 560.8792, Y 56.4939, Z -2.1667, A 0.000, B 0.000, C 0.000 }
gfCNCPoint1[19740] = {X 559.3427, Y 56.1777, Z -2.1667, A 0.000, B 0.000, C 0.000 }
gfCNCPoint1[19741] = {X 557.8630, Y 55.6570, Z -2.1667, A 0.000, B 0.000, C 0.000 }
gfCNCPoint1[19742] = {X 556.4670, Y 54.9414, Z -2.1667, A 0.000, B 0.000, C 0.000 }
gfCNCPoint1[19743] = {X 555.1803, Y 54.0440, Z -2.1667, A 0.000, B 0.000, C 0.000 }
gfCNCPoint1[19744] = {X 554.0265, Y 52.9812, Z -2.1667, A 0.000, B 0.000, C 0.000 }
gfCNCPoint1[19745] = {X 553.0266, Y 51.7725, Z -2.1667, A 0.000, B 0.000, C 0.000 }
gfCNCPoint1[19746] = {X 552.1989, Y 50.4399, Z -2.1667, A 0.000, B 0.000, C 0.000 }
gfCNCPoint1[19747] = {X 551.5587, Y 49.0078, Z -2.1667, A 0.000, B 0.000, C 0.000 }
gfCNCPoint1[19748] = {X 551.1636, Y 47.7031, Z -2.1667, A 0.000, B 0.000, C 0.000 }
gfCNCPoint1[19749] = {X 550.9244, Y 46.3609, Z -2.1667, A 0.000, B 0.000, C 0.000 }
gfCNCPoint1[19750] = {X 550.8443, Y 45.0000, Z -2.1667, A 0.000, B 0.000, C 0.000 }
gfCNCPoint1[19751] = {X 550.8443, Y 44.0525, Z -2.1667, A 0.000, B 0.000, C 0.000 }
gfCNCPoint1[19752] = {X 550.9573, Y 42.4677, Z -2.1667, A 0.000, B 0.000, C 0.000 }
gfCNCPoint1[19753] = {X 551.2851, Y 40.9130, Z -2.1667, A 0.000, B 0.000, C 0.000 }
gfCNCPoint1[19754] = {X 551.8216, Y 39.4174, Z -2.1667, A 0.000, B 0.000, C 0.000 }
gfCNCPoint1[19755] = {X 549.6231, Y 38.4547, Z -2.1667, A 0.000, B 0.000, C 0.000 }
gfCNCPoint1[19756] = {X 549.7925, Y 38.0827, Z -2.1667, A 0.000, B 0.000, C 0.000 }
gfCNCPoint1[19757] = {X 549.9727, Y 37.7157, Z -2.1667, A 0.000, B 0.000, C 0.000 }
gfCNCPoint1[19758] = {X 549.9727, Y 16.9496, Z -2.1667, A 0.000, B 0.000, C 0.000 }
gfCNCPoint1[19759] = {X 549.8029, Y 17.1989, Z -2.1667, A 0.000, B 0.000, C 0.000 }
gfCNCPoint1[19760] = {X 549.6229, Y 17.4411, Z -2.1667, A 0.000, B 0.000, C 0.000 }
gfCNCPoint1[19761] = {X 549.6231, Y 38.4547, Z -2.1667, A 0.000, B 0.000, C 0.000 }
gfCNCPoint1[19762] = {X 551.8216, Y 39.4174, Z -2.1667, A 0.000, B 0.000, C 0.000 }
gfCNCPoint1[19763] = {X 552.0826, Y 38.8616, Z -2.1667, A 0.000, B 0.000, C 0.000 }
gfCNCPoint1[19764] = {X 552.3727, Y 38.3203, Z -2.1667, A 0.000, B 0.000, C 0.000 }
gfCNCPoint1[19765] = {X 552.3727, Y 11.6893, Z -2.1667, A 0.000, B 0.000, C 0.000 }
gfCNCPoint1[19766] = {X 551.6709, Y 10.2346, Z -2.1667, A 0.000, B 0.000, C 0.000 }
gfCNCPoint1[19767] = {X 551.1781, Y 8.6966, Z -2.1667, A 0.000, B 0.000, C 0.000 }
gfCNCPoint1[19768] = {X 550.9036, Y 7.1051, Z -2.1667, A 0.000, B 0.000, C 0.000 }
gfCNCPoint1[19769] = {X 524.2928, Y 7.1051, Z -2.1667, A 0.000, B 0.000, C 0.000 }
gfCNCPoint1[19770] = {X 524.3790, Y 7.2069, Z -2.1667, A 0.000, B 0.000, C 0.000 }
gfCNCPoint1[19771] = {X 524.4623, Y 7.3110, Z -2.1667, A 0.000, B 0.000, C 0.000 }
gfCNCPoint1[19772] = {X 543.7426, Y 7.3116, Z -2.1667, A 0.000, B 0.000, C 0.000 }
gfCNCPoint1[19773] = {X 544.7118, Y 7.3837, Z -2.1667, A 0.000, B 0.000, C 0.000 }
gfCNCPoint1[19774] = {X 545.6474, Y 7.6462, Z -2.1667, A 0.000, B 0.000, C 0.000 }
gfCNCPoint1[19775] = {X 546.5126, Y 8.0888, Z -2.1667, A 0.000, B 0.000, C 0.000 }
gfCNCPoint1[19776] = {X 547.2731, Y 8.6938, Z -2.1667, A 0.000, B 0.000, C 0.000 }
gfCNCPoint1[19777] = {X 547.8987, Y 9.4374, Z -2.1667, A 0.000, B 0.000, C 0.000 }
gfCNCPoint1[19778] = {X 548.3648, Y 10.2902, Z -2.1667, A 0.000, B 0.000, C 0.000 }
gfCNCPoint1[19779] = {X 548.6528, Y 11.2183, Z -2.1667, A 0.000, B 0.000, C 0.000 }
gfCNCPoint1[19780] = {X 548.7514, Y 12.1851, Z -2.1667, A 0.000, B 0.000, C 0.000 }
gfCNCPoint1[19781] = {X 548.7512, Y 13.0282, Z -2.1667, A 0.000, B 0.000, C 0.000 }
gfCNCPoint1[19782] = {X 548.6549, Y 13.9437, Z -2.1667, A 0.000, B 0.000, C 0.000 }
gfCNCPoint1[19783] = {X 548.3885, Y 14.8248, Z -2.1667, A 0.000, B 0.000, C 0.000 }
gfCNCPoint1[19784] = {X 547.9613, Y 15.6403, Z -2.1667, A 0.000, B 0.000, C 0.000 }
gfCNCPoint1[19785] = {X 547.6183, Y 16.1046, Z -2.1667, A 0.000, B 0.000, C 0.000 }
gfCNCPoint1[19786] = {X 547.2229, Y 16.5251, Z -2.1667, A 0.000, B 0.000, C 0.000 }
gfCNCPoint1[19787] = {X 547.2231, Y 40.6619, Z -2.1667, A 0.000, B 0.000, C 0.000 }
gfCNCPoint1[19788] = {X 547.8648, Y 41.4039, Z -2.1667, A 0.000, B 0.000, C 0.000 }
gfCNCPoint1[19789] = {X 548.3451, Y 42.2593, Z -2.1667, A 0.000, B 0.000, C 0.000 }
gfCNCPoint1[19790] = {X 548.6446, Y 43.1935, Z -2.1667, A 0.000, B 0.000, C 0.000 }
gfCNCPoint1[19791] = {X 548.7513, Y 44.1687, Z -2.1667, A 0.000, B 0.000, C 0.000 }
gfCNCPoint1[19792] = {X 548.7514, Y 45.0017, Z -2.1667, A 0.000, B 0.000, C 0.000 }
gfCNCPoint1[19793] = {X 548.6695, Y 45.8828, Z -2.1667, A 0.000, B 0.000, C 0.000 }
gfCNCPoint1[19794] = {X 548.4299, Y 46.7347, Z -2.1667, A 0.000, B 0.000, C 0.000 }
gfCNCPoint1[19795] = {X 548.0406, Y 47.5294, Z -2.1667, A 0.000, B 0.000, C 0.000 }
gfCNCPoint1[19796] = {X 547.5143, Y 48.2408, Z -2.1667, A 0.000, B 0.000, C 0.000 }
gfCNCPoint1[19797] = {X 546.7287, Y 48.9503, Z -2.1667, A 0.000, B 0.000, C 0.000 }
gfCNCPoint1[19798] = {X 545.8087, Y 49.4739, Z -2.1667, A 0.000, B 0.000, C 0.000 }
gfCNCPoint1[19799] = {X 544.7975, Y 49.7870, Z -2.1667, A 0.000, B 0.000, C 0.000 }
gfCNCPoint1[19800] = {X 543.7426, Y 49.8749, Z -2.1667, A 0.000, B 0.000, C 0.000 }
gfCNCPoint1[19801] = {X 524.3231, Y 49.8755, Z -2.1667, A 0.000, B 0.000, C 0.000 }
gfCNCPoint1[19802] = {X 523.7104, Y 50.5144, Z -2.1667, A 0.000, B 0.000, C 0.000 }
gfCNCPoint1[19803] = {X 522.9953, Y 51.0363, Z -2.1667, A 0.000, B 0.000, C 0.000 }
gfCNCPoint1[19804] = {X 522.1998, Y 51.4249, Z -2.1667, A 0.000, B 0.000, C 0.000 }
gfCNCPoint1[19805] = {X 521.3487, Y 51.6684, Z -2.1667, A 0.000, B 0.000, C 0.000 }
gfCNCPoint1[19806] = {X 520.4681, Y 51.7591, Z -2.1667, A 0.000, B 0.000, C 0.000 }
gfCNCPoint1[19807] = {X 519.7998, Y 51.7591, Z -2.1667, A 0.000, B 0.000, C 0.000 }
gfCNCPoint1[19808] = {X 518.8477, Y 51.6654, Z -2.1667, A 0.000, B 0.000, C 0.000 }
gfCNCPoint1[19809] = {X 517.9323, Y 51.3877, Z -2.1667, A 0.000, B 0.000, C 0.000 }
gfCNCPoint1[19810] = {X 517.0886, Y 50.9367, Z -2.1667, A 0.000, B 0.000, C 0.000 }
gfCNCPoint1[19811] = {X 516.3491, Y 50.3298, Z -2.1667, A 0.000, B 0.000, C 0.000 }
gfCNCPoint1[19812] = {X 515.7422, Y 49.5903, Z -2.1667, A 0.000, B 0.000, C 0.000 }
gfCNCPoint1[19813] = {X 515.2912, Y 48.7466, Z -2.1667, A 0.000, B 0.000, C 0.000 }
gfCNCPoint1[19814] = {X 515.0135, Y 47.8312, Z -2.1667, A 0.000, B 0.000, C 0.000 }
gfCNCPoint1[19815] = {X 514.9198, Y 46.8791, Z -2.1667, A 0.000, B 0.000, C 0.000 }
gfCNCPoint1[19816] = {X 514.9198, Y 39.9011, Z -2.1667, A 0.000, B 0.000, C 0.000 }
gfCNCPoint1[19817] = {X 515.0197, Y 38.9186, Z -2.1667, A 0.000, B 0.000, C 0.000 }
gfCNCPoint1[19818] = {X 515.3154, Y 37.9764, Z -2.1667, A 0.000, B 0.000, C 0.000 }
gfCNCPoint1[19819] = {X 515.7947, Y 37.1129, Z -2.1667, A 0.000, B 0.000, C 0.000 }
gfCNCPoint1[19820] = {X 516.4381, Y 36.3637, Z -2.1667, A 0.000, B 0.000, C 0.000 }
gfCNCPoint1[19821] = {X 517.2191, Y 35.7593, Z -2.1667, A 0.000, B 0.000, C 0.000 }
gfCNCPoint1[19822] = {X 518.1058, Y 35.3245, Z -2.1667, A 0.000, B 0.000, C 0.000 }
gfCNCPoint1[19823] = {X 519.0619, Y 35.0772, Z -2.1667, A 0.000, B 0.000, C 0.000 }
gfCNCPoint1[19824] = {X 519.4084, Y 35.0368, Z -2.1667, A 0.000, B 0.000, C 0.000 }
gfCNCPoint1[19825] = {X 519.7568, Y 35.0213, Z -2.1667, A 0.000, B 0.000, C 0.000 }
gfCNCPoint1[19826] = {X 520.5345, Y 35.0216, Z -2.1667, A 0.000, B 0.000, C 0.000 }
gfCNCPoint1[19827] = {X 521.4086, Y 35.1126, Z -2.1667, A 0.000, B 0.000, C 0.000 }
gfCNCPoint1[19828] = {X 522.2523, Y 35.3589, Z -2.1667, A 0.000, B 0.000, C 0.000 }
gfCNCPoint1[19829] = {X 523.0381, Y 35.7526, Z -2.1667, A 0.000, B 0.000, C 0.000 }
gfCNCPoint1[19830] = {X 523.7405, Y 36.2808, Z -2.1667, A 0.000, B 0.000, C 0.000 }
gfCNCPoint1[19831] = {X 524.3368, Y 36.9265, Z -2.1667, A 0.000, B 0.000, C 0.000 }
gfCNCPoint1[19832] = {X 534.0719, Y 36.9270, Z -2.1667, A 0.000, B 0.000, C 0.000 }
gfCNCPoint1[19833] = {X 534.0719, Y 34.5247, Z -2.1667, A 0.000, B 0.000, C 0.000 }
gfCNCPoint1[19834] = {X 530.3969, Y 34.5243, Z -2.1667, A 0.000, B 0.000, C 0.000 }
gfCNCPoint1[19835] = {X 529.7970, Y 35.1731, Z -2.1667, A 0.000, B 0.000, C 0.000 }
gfCNCPoint1[19836] = {X 529.0899, Y 35.7032, Z -2.1667, A 0.000, B 0.000, C 0.000 }
gfCNCPoint1[19837] = {X 528.2988, Y 36.0970, Z -2.1667, A 0.000, B 0.000, C 0.000 }
gfCNCPoint1[19838] = {X 527.4496, Y 36.3417, Z -2.1667, A 0.000, B 0.000, C 0.000 }
gfCNCPoint1[19839] = {X 526.5703, Y 36.4293, Z -2.1667, A 0.000, B 0.000, C 0.000 }
gfCNCPoint1[19840] = {X 525.8868, Y 36.4294, Z -2.1667, A 0.000, B 0.000, C 0.000 }
gfCNCPoint1[19841] = {X 524.9094, Y 36.3306, Z -2.1667, A 0.000, B 0.000, C 0.000 }
gfCNCPoint1[19842] = {X 523.9717, Y 36.0380, Z -2.1667, A 0.000, B 0.000, C 0.000 }
gfCNCPoint1[19843] = {X 523.1116, Y 35.5636, Z -2.1667, A 0.000, B 0.000, C 0.000 }
gfCNCPoint1[19844] = {X 522.3639, Y 34.9265, Z -2.1667, A 0.000, B 0.000, C 0.000 }
gfCNCPoint1[19845] = {X 521.7590, Y 34.1525, Z -2.1667, A 0.000, B 0.000, C 0.000 }
gfCNCPoint1[19846] = {X 521.3213, Y 33.2731, Z -2.1667, A 0.000, B 0.000, C 0.000 }
gfCNCPoint1[19847] = {X 521.0686, Y 32.3239, Z -2.1667, A 0.000, B 0.000, C 0.000 }
gfCNCPoint1[19848] = {X 521.0222, Y 31.9379, Z -2.1667, A 0.000, B 0.000, C 0.000 }
gfCNCPoint1[19849] = {X 521.0068, Y 31.5495, Z -2.1667, A 0.000, B 0.000, C 0.000 }
gfCNCPoint1[19850] = {X 521.0076, Y 24.4815, Z -2.1667, A 0.000, B 0.000, C 0.000 }
gfCNCPoint1[19851] = {X 521.0984, Y 23.6300, Z -2.1667, A 0.000, B 0.000, C 0.000 }
gfCNCPoint1[19852] = {X 521.3368, Y 22.8074, Z -2.1667, A 0.000, B 0.000, C 0.000 }
gfCNCPoint1[19853] = {X 521.7152, Y 22.0391, Z -2.1667, A 0.000, B 0.000, C 0.000 }
gfCNCPoint1[19854] = {X 521.1864, Y 22.1316, Z -2.1667, A 0.000, B 0.000, C 0.000 }
gfCNCPoint1[19855] = {X 520.6505, Y 22.1656, Z -2.1667, A 0.000, B 0.000, C 0.000 }
gfCNCPoint1[19856] = {X 519.9691, Y 22.1657, Z -2.1667, A 0.000, B 0.000, C 0.000 }
gfCNCPoint1[19857] = {X 519.5109, Y 22.1442, Z -2.1667, A 0.000, B 0.000, C 0.000 }
gfCNCPoint1[19858] = {X 519.0567, Y 22.0797, Z -2.1667, A 0.000, B 0.000, C 0.000 }
gfCNCPoint1[19859] = {X 518.1336, Y 21.8074, Z -2.1667, A 0.000, B 0.000, C 0.000 }
gfCNCPoint1[19860] = {X 517.2820, Y 21.3592, Z -2.1667, A 0.000, B 0.000, C 0.000 }
gfCNCPoint1[19861] = {X 516.5348, Y 20.7527, Z -2.1667, A 0.000, B 0.000, C 0.000 }
gfCNCPoint1[19862] = {X 515.9212, Y 20.0113, Z -2.1667, A 0.000, B 0.000, C 0.000 }
gfCNCPoint1[19863] = {X 515.4650, Y 19.1639, Z -2.1667, A 0.000, B 0.000, C 0.000 }
gfCNCPoint1[19864] = {X 515.1840, Y 18.2434, Z -2.1667, A 0.000, B 0.000, C 0.000 }
gfCNCPoint1[19865] = {X 515.0891, Y 17.2857, Z -2.1667, A 0.000, B 0.000, C 0.000 }
gfCNCPoint1[19866] = {X 515.0891, Y 10.3077, Z -2.1667, A 0.000, B 0.000, C 0.000 }
gfCNCPoint1[19867] = {X 515.0965, Y 10.0383, Z -2.1667, A 0.000, B 0.000, C 0.000 }
gfCNCPoint1[19868] = {X 515.1189, Y 9.7697, Z -2.1667, A 0.000, B 0.000, C 0.000 }
gfCNCPoint1[19869] = {X 515.3251, Y 8.8084, Z -2.1667, A 0.000, B 0.000, C 0.000 }
gfCNCPoint1[19870] = {X 515.7198, Y 7.9081, Z -2.1667, A 0.000, B 0.000, C 0.000 }
gfCNCPoint1[19871] = {X 516.2870, Y 7.1051, Z -2.1667, A 0.000, B 0.000, C 0.000 }
gfCNCPoint1[19872] = {X 516.6492, Y 7.4201, Z -2.1667, A 0.000, B 0.000, C 0.000 }
gfCNCPoint1[19873] = {X 517.3373, Y 6.7816, Z -2.1667, A 0.000, B 0.000, C 0.000 }
gfCNCPoint1[19874] = {X 518.1451, Y 6.3036, Z -2.1667, A 0.000, B 0.000, C 0.000 }
gfCNCPoint1[19875] = {X 519.0359, Y 6.0078, Z -2.1667, A 0.000, B 0.000, C 0.000 }
gfCNCPoint1[19876] = {X 519.9692, Y 5.9077, Z -2.1667, A 0.000, B 0.000, C 0.000 }
gfCNCPoint1[19877] = {X 520.6509, Y 5.9079, Z -2.1667, A 0.000, B 0.000, C 0.000 }
gfCNCPoint1[19878] = {X 521.4835, Y 5.9951, Z -2.1667, A 0.000, B 0.000, C 0.000 }
gfCNCPoint1[19879] = {X 522.2845, Y 6.2385, Z -2.1667, A 0.000, B 0.000, C 0.000 }
gfCNCPoint1[19880] = {X 523.0249, Y 6.6291, Z -2.1667, A 0.000, B 0.000, C 0.000 }
gfCNCPoint1[19881] = {X 523.6780, Y 7.1530, Z -2.1667, A 0.000, B 0.000, C 0.000 }
gfCNCPoint1[19882] = {X 524.2200, Y 7.7910, Z -2.1667, A 0.000, B 0.000, C 0.000 }
gfCNCPoint1[19883] = {X 543.7489, Y 7.7916, Z -2.1667, A 0.000, B 0.000, C 0.000 }
gfCNCPoint1[19884] = {X 544.7469, Y 7.8789, Z -2.1667, A 0.000, B 0.000, C 0.000 }
gfCNCPoint1[19885] = {X 545.6994, Y 8.1895, Z -2.1667, A 0.000, B 0.000, C 0.000 }
gfCNCPoint1[19886] = {X 546.5570, Y 8.7072, Z -2.1667, A 0.000, B 0.000, C 0.000 }
gfCNCPoint1[19887] = {X 547.2755, Y 9.4054, Z -2.1667, A 0.000, B 0.000, C 0.000 }
gfCNCPoint1[19888] = {X 547.8177, Y 10.2478, Z -2.1667, A 0.000, B 0.000, C 0.000 }
gfCNCPoint1[19889] = {X 548.1555, Y 11.1910, Z -2.1667, A 0.000, B 0.000, C 0.000 }
gfCNCPoint1[19890] = {X 548.2714, Y 12.1861, Z -2.1667, A 0.000, B 0.000, C 0.000 }
gfCNCPoint1[19891] = {X 548.2712, Y 13.0233, Z -2.1667, A 0.000, B 0.000, C 0.000 }
gfCNCPoint1[19892] = {X 548.1628, Y 13.9497, Z -2.1667, A 0.000, B 0.000, C 0.000 }
gfCNCPoint1[19893] = {X 547.8616, Y 14.8324, Z -2.1667, A 0.000, B 0.000, C 0.000 }
gfCNCPoint1[19894] = {X 547.3811, Y 15.6317, Z -2.1667, A 0.000, B 0.000, C 0.000 }
gfCNCPoint1[19895] = {X 546.7429, Y 16.3119, Z -2.1667, A 0.000, B 0.000, C 0.000 }
gfCNCPoint1[19896] = {X 546.7431, Y 40.8751, Z -2.1667, A 0.000, B 0.000, C 0.000 }
gfCNCPoint1[19897] = {X 547.3881, Y 41.5643, Z -2.1667, A 0.000, B 0.000, C 0.000 }
gfCNCPoint1[19898] = {X 547.8712, Y 42.3752, Z -2.1667, A 0.000, B 0.000, C 0.000 }
gfCNCPoint1[19899] = {X 548.1702, Y 43.2705, Z -2.1667, A 0.000, B 0.000, C 0.000 }
gfCNCPoint1[19900] = {X 548.2714, Y 44.2089, Z -2.1667, A 0.000, B 0.000, C 0.000 }
gfCNCPoint1[19901] = {X 548.2714, Y 45.0008, Z -2.1667, A 0.000, B 0.000, C 0.000 }
gfCNCPoint1[19902] = {X 548.1555, Y 45.9958, Z -2.1667, A 0.000, B 0.000, C 0.000 }
gfCNCPoint1[19903] = {X 547.8177, Y 46.9390, Z -2.1667, A 0.000, B 0.000, C 0.000 }
gfCNCPoint1[19904] = {X 547.2755, Y 47.7814, Z -2.1667, A 0.000, B 0.000, C 0.000 }
gfCNCPoint1[19905] = {X 546.5570, Y 48.4795, Z -2.1667, A 0.000, B 0.000, C 0.000 }
gfCNCPoint1[19906] = {X 545.6993, Y 48.9972, Z -2.1667, A 0.000, B 0.000, C 0.000 }
gfCNCPoint1[19907] = {X 544.7469, Y 49.3077, Z -2.1667, A 0.000, B 0.000, C 0.000 }
gfCNCPoint1[19908] = {X 543.7489, Y 49.3949, Z -2.1667, A 0.000, B 0.000, C 0.000 }
gfCNCPoint1[19909] = {X 524.0858, Y 49.3955, Z -2.1667, A 0.000, B 0.000, C 0.000 }
gfCNCPoint1[19910] = {X 523.5291, Y 50.0305, Z -2.1667, A 0.000, B 0.000, C 0.000 }
gfCNCPoint1[19911] = {X 522.8648, Y 50.5520, Z -2.1667, A 0.000, B 0.000, C 0.000 }
gfCNCPoint1[19912] = {X 522.1157, Y 50.9420, Z -2.1667, A 0.000, B 0.000, C 0.000 }
gfCNCPoint1[19913] = {X 521.3076, Y 51.1872, Z -2.1667, A 0.000, B 0.000, C 0.000 }
gfCNCPoint1[19914] = {X 520.4681, Y 51.2791, Z -2.1667, A 0.000, B 0.000, C 0.000 }
gfCNCPoint1[19915] = {X 519.7998, Y 51.2791, Z -2.1667, A 0.000, B 0.000, C 0.000 }
gfCNCPoint1[19916] = {X 518.8207, Y 51.1688, Z -2.1667, A 0.000, B 0.000, C 0.000 }
gfCNCPoint1[19917] = {X 517.8907, Y 50.8434, Z -2.1667, A 0.000, B 0.000, C 0.000 }
gfCNCPoint1[19918] = {X 517.0564, Y 50.3192, Z -2.1667, A 0.000, B 0.000, C 0.000 }
gfCNCPoint1[19919] = {X 516.3597, Y 49.6225, Z -2.1667, A 0.000, B 0.000, C 0.000 }
gfCNCPoint1[19920] = {X 515.8355, Y 48.7882, Z -2.1667, A 0.000, B 0.000, C 0.000 }
gfCNCPoint1[19921] = {X 515.5101, Y 47.8582, Z -2.1667, A 0.000, B 0.000, C 0.000 }
gfCNCPoint1[19922] = {X 515.3998, Y 46.8791, Z -2.1667, A 0.000, B 0.000, C 0.000 }
gfCNCPoint1[19923] = {X 515.3998, Y 39.9011, Z -2.1667, A 0.000, B 0.000, C 0.000 }
gfCNCPoint1[19924] = {X 515.5101, Y 38.9220, Z -2.1667, A 0.000, B 0.000, C 0.000 }
gfCNCPoint1[19925] = {X 515.8355, Y 37.9920, Z -2.1667, A 0.000, B 0.000, C 0.000 }
gfCNCPoint1[19926] = {X 516.3597, Y 37.1577, Z -2.1667, A 0.000, B 0.000, C 0.000 }
gfCNCPoint1[19927] = {X 517.0565, Y 36.4610, Z -2.1667, A 0.000, B 0.000, C 0.000 }
gfCNCPoint1[19928] = {X 517.8907, Y 35.9368, Z -2.1667, A 0.000, B 0.000, C 0.000 }
gfCNCPoint1[19929] = {X 518.8208, Y 35.6114, Z -2.1667, A 0.000, B 0.000, C 0.000 }
gfCNCPoint1[19930] = {X 519.7999, Y 35.5011, Z -2.1667, A 0.000, B 0.000, C 0.000 }
gfCNCPoint1[19931] = {X 520.5280, Y 35.5015, Z -2.1667, A 0.000, B 0.000, C 0.000 }
gfCNCPoint1[19932] = {X 521.3616, Y 35.5928, Z -2.1667, A 0.000, B 0.000, C 0.000 }
gfCNCPoint1[19933] = {X 522.1628, Y 35.8405, Z -2.1667, A 0.000, B 0.000, C 0.000 }
gfCNCPoint1[19934] = {X 522.9024, Y 36.2358, Z -2.1667, A 0.000, B 0.000, C 0.000 }
gfCNCPoint1[19935] = {X 523.5536, Y 36.7642, Z -2.1667, A 0.000, B 0.000, C 0.000 }
gfCNCPoint1[19936] = {X 524.0927, Y 37.4065, Z -2.1667, A 0.000, B 0.000, C 0.000 }
gfCNCPoint1[19937] = {X 534.5519, Y 37.4071, Z -2.1667, A 0.000, B 0.000, C 0.000 }
gfCNCPoint1[19938] = {X 534.5519, Y 34.0447, Z -2.1667, A 0.000, B 0.000, C 0.000 }
gfCNCPoint1[19939] = {X 530.1528, Y 34.0442, Z -2.1667, A 0.000, B 0.000, C 0.000 }
gfCNCPoint1[19940] = {X 529.6051, Y 34.6949, Z -2.1667, A 0.000, B 0.000, C 0.000 }
gfCNCPoint1[19941] = {X 528.9425, Y 35.2281, Z -2.1667, A 0.000, B 0.000, C 0.000 }
gfCNCPoint1[19942] = {X 528.1897, Y 35.6238, Z -2.1667, A 0.000, B 0.000, C 0.000 }
gfCNCPoint1[19943] = {X 527.3748, Y 35.8673, Z -2.1667, A 0.000, B 0.000, C 0.000 }
gfCNCPoint1[19944] = {X 526.5283, Y 35.9495, Z -2.1667, A 0.000, B 0.000, C 0.000 }
gfCNCPoint1[19945] = {X 525.8868, Y 35.9495, Z -2.1667, A 0.000, B 0.000, C 0.000 }
gfCNCPoint1[19946] = {X 524.9077, Y 35.8391, Z -2.1667, A 0.000, B 0.000, C 0.000 }
gfCNCPoint1[19947] = {X 523.9777, Y 35.5137, Z -2.1667, A 0.000, B 0.000, C 0.000 }
gfCNCPoint1[19948] = {X 523.1434, Y 34.9895, Z -2.1667, A 0.000, B 0.000, C 0.000 }
gfCNCPoint1[19949] = {X 522.4467, Y 34.2928, Z -2.1667, A 0.000, B 0.000, C 0.000 }
gfCNCPoint1[19950] = {X 521.9225, Y 33.4585, Z -2.1667, A 0.000, B 0.000, C 0.000 }
gfCNCPoint1[19951] = {X 521.5971, Y 32.5285, Z -2.1667, A 0.000, B 0.000, C 0.000 }
gfCNCPoint1[19952] = {X 521.4868, Y 31.5495, Z -2.1667, A 0.000, B 0.000, C 0.000 }
gfCNCPoint1[19953] = {X 521.4868, Y 24.5714, Z -2.1667, A 0.000, B 0.000, C 0.000 }
gfCNCPoint1[19954] = {X 521.5971, Y 23.5923, Z -2.1667, A 0.000, B 0.000, C 0.000 }
gfCNCPoint1[19955] = {X 521.9225, Y 22.6623, Z -2.1667, A 0.000, B 0.000, C 0.000 }
gfCNCPoint1[19956] = {X 522.4467, Y 21.8281, Z -2.1667, A 0.000, B 0.000, C 0.000 }
gfCNCPoint1[19957] = {X 523.1434, Y 21.1314, Z -2.1667, A 0.000, B 0.000, C 0.000 }
gfCNCPoint1[19958] = {X 523.9777, Y 20.6072, Z -2.1667, A 0.000, B 0.000, C 0.000 }
gfCNCPoint1[19959] = {X 524.9077, Y 20.2817, Z -2.1667, A 0.000, B 0.000, C 0.000 }
gfCNCPoint1[19960] = {X 525.8868, Y 20.1714, Z -2.1667, A 0.000, B 0.000, C 0.000 }
gfCNCPoint1[19961] = {X 526.5702, Y 20.1716, Z -2.1667, A 0.000, B 0.000, C 0.000 }
gfCNCPoint1[19962] = {X 527.2684, Y 20.2341, Z -2.1667, A 0.000, B 0.000, C 0.000 }
gfCNCPoint1[19963] = {X 527.9478, Y 20.4066, Z -2.1667, A 0.000, B 0.000, C 0.000 }
gfCNCPoint1[19964] = {X 528.5912, Y 20.6849, Z -2.1667, A 0.000, B 0.000, C 0.000 }
gfCNCPoint1[19965] = {X 528.8162, Y 20.2609, Z -2.1667, A 0.000, B 0.000, C 0.000 }
gfCNCPoint1[19966] = {X 534.0719, Y 20.2612, Z -2.1667, A 0.000, B 0.000, C 0.000 }
gfCNCPoint1[19967] = {X 534.0719, Y 21.5750, Z -2.1667, A 0.000, B 0.000, C 0.000 }
gfCNCPoint1[19968] = {X 530.3799, Y 21.5747, Z -2.1667, A 0.000, B 0.000, C 0.000 }
gfCNCPoint1[19969] = {X 529.6676, Y 20.8351, Z -2.1667, A 0.000, B 0.000, C 0.000 }
gfCNCPoint1[19970] = {X 528.8162, Y 20.2609, Z -2.1667, A 0.000, B 0.000, C 0.000 }
gfCNCPoint1[19971] = {X 528.5912, Y 20.6849, Z -2.1667, A 0.000, B 0.000, C 0.000 }
gfCNCPoint1[19972] = {X 529.1769, Y 21.0578, Z -2.1667, A 0.000, B 0.000, C 0.000 }
gfCNCPoint1[19973] = {X 529.6967, Y 21.5182, Z -2.1667, A 0.000, B 0.000, C 0.000 }
gfCNCPoint1[19974] = {X 530.1376, Y 22.0547, Z -2.1667, A 0.000, B 0.000, C 0.000 }
gfCNCPoint1[19975] = {X 534.5519, Y 22.0550, Z -2.1667, A 0.000, B 0.000, C 0.000 }
gfCNCPoint1[19976] = {X 534.5519, Y 19.7812, Z -2.1667, A 0.000, B 0.000, C 0.000 }
gfCNCPoint1[19977] = {X 524.2350, Y 19.7807, Z -2.1667, A 0.000, B 0.000, C 0.000 }
gfCNCPoint1[19978] = {X 523.6873, Y 20.4313, Z -2.1667, A 0.000, B 0.000, C 0.000 }
gfCNCPoint1[19979] = {X 523.0247, Y 20.9644, Z -2.1667, A 0.000, B 0.000, C 0.000 }
gfCNCPoint1[19980] = {X 522.2720, Y 21.3601, Z -2.1667, A 0.000, B 0.000, C 0.000 }
gfCNCPoint1[19981] = {X 521.4571, Y 21.6035, Z -2.1667, A 0.000, B 0.000, C 0.000 }
gfCNCPoint1[19982] = {X 520.6107, Y 21.6857, Z -2.1667, A 0.000, B 0.000, C 0.000 }
gfCNCPoint1[19983] = {X 519.9691, Y 21.6857, Z -2.1667, A 0.000, B 0.000, C 0.000 }
gfCNCPoint1[19984] = {X 518.9900, Y 21.5754, Z -2.1667, A 0.000, B 0.000, C 0.000 }
gfCNCPoint1[19985] = {X 518.0600, Y 21.2500, Z -2.1667, A 0.000, B 0.000, C 0.000 }
gfCNCPoint1[19986] = {X 517.2257, Y 20.7258, Z -2.1667, A 0.000, B 0.000, C 0.000 }
gfCNCPoint1[19987] = {X 516.5290, Y 20.0291, Z -2.1667, A 0.000, B 0.000, C 0.000 }
gfCNCPoint1[19988] = {X 516.0048, Y 19.1948, Z -2.1667, A 0.000, B 0.000, C 0.000 }
gfCNCPoint1[19989] = {X 515.6794, Y 18.2648, Z -2.1667, A 0.000, B 0.000, C 0.000 }
gfCNCPoint1[19990] = {X 515.5691, Y 17.2857, Z -2.1667, A 0.000, B 0.000, C 0.000 }
gfCNCPoint1[19991] = {X 515.5691, Y 10.3077, Z -2.1667, A 0.000, B 0.000, C 0.000 }
gfCNCPoint1[19992] = {X 515.6394, Y 9.5244, Z -2.1667, A 0.000, B 0.000, C 0.000 }
gfCNCPoint1[19993] = {X 515.8480, Y 8.7662, Z -2.1667, A 0.000, B 0.000, C 0.000 }
gfCNCPoint1[19994] = {X 516.1882, Y 8.0572, Z -2.1667, A 0.000, B 0.000, C 0.000 }
gfCNCPoint1[19995] = {X 516.6492, Y 7.4201, Z -2.1667, A 0.000, B 0.000, C 0.000 }
gfCNCPoint1[19996] = {X 516.2870, Y 7.1051, Z -2.1667, A 0.000, B 0.000, C 0.000 }
gfCNCPoint1[19997] = {X 370.1019, Y 7.1051, Z -2.1667, A 0.000, B 0.000, C 0.000 }
gfCNCPoint1[19998] = {X 371.1255, Y 8.7920, Z -2.1667, A 0.000, B 0.000, C 0.000 }
gfCNCPoint1[19999] = {X 372.0363, Y 10.5425, Z -2.1667, A 0.000, B 0.000, C 0.000 }
gfCNCPoint1[20000] = {X 372.9320, Y 12.6056, Z -2.1667, A 0.000, B 0.000, C 0.000 }
gfCNCPoint1[20001] = {X 373.6710, Y 14.7298, Z -2.1667, A 0.000, B 0.000, C 0.000 }
gfCNCPoint1[20002] = {X 374.2492, Y 16.9033, Z -2.1667, A 0.000, B 0.000, C 0.000 }
gfCNCPoint1[20003] = {X 374.7349, Y 19.4658, Z -2.1667, A 0.000, B 0.000, C 0.000 }
gfCNCPoint1[20004] = {X 375.0389, Y 22.0561, Z -2.1667, A 0.000, B 0.000, C 0.000 }
gfCNCPoint1[20005] = {X 375.1597, Y 24.6614, Z -2.1667, A 0.000, B 0.000, C 0.000 }
gfCNCPoint1[20006] = {X 375.0965, Y 27.2687, Z -2.1667, A 0.000, B 0.000, C 0.000 }
gfCNCPoint1[20007] = {X 374.8498, Y 29.8651, Z -2.1667, A 0.000, B 0.000, C 0.000 }
gfCNCPoint1[20008] = {X 374.4208, Y 32.4377, Z -2.1667, A 0.000, B 0.000, C 0.000 }
gfCNCPoint1[20009] = {X 373.7830, Y 34.9995, Z -2.1667, A 0.000, B 0.000, C 0.000 }
gfCNCPoint1[20010] = {X 372.9215, Y 37.4949, Z -2.1667, A 0.000, B 0.000, C 0.000 }
gfCNCPoint1[20011] = {X 371.8431, Y 39.9046, Z -2.1667, A 0.000, B 0.000, C 0.000 }
gfCNCPoint1[20012] = {X 370.5561, Y 42.2097, Z -2.1667, A 0.000, B 0.000, C 0.000 }
gfCNCPoint1[20013] = {X 369.0707, Y 44.3921, Z -2.1667, A 0.000, B 0.000, C 0.000 }
gfCNCPoint1[20014] = {X 369.0319, Y 44.4442, Z -2.1667, A 0.000, B 0.000, C 0.000 }
gfCNCPoint1[20015] = {X 368.9931, Y 44.4963, Z -2.1667, A 0.000, B 0.000, C 0.000 }
gfCNCPoint1[20016] = {X 367.4731, Y 46.3511, Z -2.1667, A 0.000, B 0.000, C 0.000 }
gfCNCPoint1[20017] = {X 365.7975, Y 48.0667, Z -2.1667, A 0.000, B 0.000, C 0.000 }
gfCNCPoint1[20018] = {X 363.9791, Y 49.6300, Z -2.1667, A 0.000, B 0.000, C 0.000 }
gfCNCPoint1[20019] = {X 362.0316, Y 51.0292, Z -2.1667, A 0.000, B 0.000, C 0.000 }
gfCNCPoint1[20020] = {X 359.9697, Y 52.2537, Z -2.1667, A 0.000, B 0.000, C 0.000 }
gfCNCPoint1[20021] = {X 359.3967, Y 52.5410, Z -2.1667, A 0.000, B 0.000, C 0.000 }
gfCNCPoint1[20022] = {X 358.8174, Y 52.8150, Z -2.1667, A 0.000, B 0.000, C 0.000 }
gfCNCPoint1[20023] = {X 356.4597, Y 53.7703, Z -2.1667, A 0.000, B 0.000, C 0.000 }
gfCNCPoint1[20024] = {X 354.0251, Y 54.5075, Z -2.1667, A 0.000, B 0.000, C 0.000 }
gfCNCPoint1[20025] = {X 351.5336, Y 55.0207, Z -2.1667, A 0.000, B 0.000, C 0.000 }
gfCNCPoint1[20026] = {X 349.0059, Y 55.3056, Z -2.1667, A 0.000, B 0.000, C 0.000 }
gfCNCPoint1[20027] = {X 349.9668, Y 69.6735, Z -2.1667, A 0.000, B 0.000, C 0.000 }
gfCNCPoint1[20028] = {X 348.6527, Y 69.7409, Z -2.1667, A 0.000, B 0.000, C 0.000 }
gfCNCPoint1[20029] = {X 347.3372, Y 69.7675, Z -2.1667, A 0.000, B 0.000, C 0.000 }
gfCNCPoint1[20030] = {X 346.5718, Y 69.7762, Z -2.1667, A 0.000, B 0.000, C 0.000 }
gfCNCPoint1[20031] = {X 345.8064, Y 69.7714, Z -2.1667, A 0.000, B 0.000, C 0.000 }
gfCNCPoint1[20032] = {X 345.5896, Y 70.1910, Z -2.1667, A 0.000, B 0.000, C 0.000 }
gfCNCPoint1[20033] = {X 345.3647, Y 70.6062, Z -2.1667, A 0.000, B 0.000, C 0.000 }
gfCNCPoint1[20034] = {X 346.5802, Y 70.6171, Z -2.1667, A 0.000, B 0.000, C 0.000 }
gfCNCPoint1[20035] = {X 347.7957, Y 70.6136, Z -2.1667, A 0.000, B 0.000, C 0.000 }
gfCNCPoint1[20036] = {X 349.1270, Y 70.6194, Z -2.1667, A 0.000, B 0.000, C 0.000 }
gfCNCPoint1[20037] = {X 350.4582, Y 70.6078, Z -2.1667, A 0.000, B 0.000, C 0.000 }
gfCNCPoint1[20038] = {X 350.2073, Y 70.1433, Z -2.1667, A 0.000, B 0.000, C 0.000 }
gfCNCPoint1[20039] = {X 349.9668, Y 69.6735, Z -2.1667, A 0.000, B 0.000, C 0.000 }
gfCNCPoint1[20040] = {X 349.8066, Y 67.2788, Z -2.1667, A 0.000, B 0.000, C 0.000 }
gfCNCPoint1[20041] = {X 348.5577, Y 67.3428, Z -2.1667, A 0.000, B 0.000, C 0.000 }
gfCNCPoint1[20042] = {X 347.3074, Y 67.3676, Z -2.1667, A 0.000, B 0.000, C 0.000 }
gfCNCPoint1[20043] = {X 345.8015, Y 67.3710, Z -2.1667, A 0.000, B 0.000, C 0.000 }
gfCNCPoint1[20044] = {X 344.2964, Y 67.3194, Z -2.1667, A 0.000, B 0.000, C 0.000 }
gfCNCPoint1[20045] = {X 343.8099, Y 68.3949, Z -2.1667, A 0.000, B 0.000, C 0.000 }
gfCNCPoint1[20046] = {X 343.2658, Y 69.4423, Z -2.1667, A 0.000, B 0.000, C 0.000 }
gfCNCPoint1[20047] = {X 342.7863, Y 70.2639, Z -2.1667, A 0.000, B 0.000, C 0.000 }
gfCNCPoint1[20048] = {X 342.2714, Y 71.0638, Z -2.1667, A 0.000, B 0.000, C 0.000 }
gfCNCPoint1[20049] = {X 342.2715, Y 72.9166, Z -2.1667, A 0.000, B 0.000, C 0.000 }
gfCNCPoint1[20050] = {X 343.8000, Y 72.9723, Z -2.1667, A 0.000, B 0.000, C 0.000 }
gfCNCPoint1[20051] = {X 345.3292, Y 73.0059, Z -2.1667, A 0.000, B 0.000, C 0.000 }
gfCNCPoint1[20052] = {X 346.5611, Y 73.0170, Z -2.1667, A 0.000, B 0.000, C 0.000 }
gfCNCPoint1[20053] = {X 347.7932, Y 73.0137, Z -2.1667, A 0.000, B 0.000, C 0.000 }
gfCNCPoint1[20054] = {X 349.1440, Y 73.0194, Z -2.1667, A 0.000, B 0.000, C 0.000 }
gfCNCPoint1[20055] = {X 350.4947, Y 73.0075, Z -2.1667, A 0.000, B 0.000, C 0.000 }
gfCNCPoint1[20056] = {X 352.0278, Y 72.9729, Z -2.1667, A 0.000, B 0.000, C 0.000 }
gfCNCPoint1[20057] = {X 353.5602, Y 72.9158, Z -2.1667, A 0.000, B 0.000, C 0.000 }
gfCNCPoint1[20058] = {X 353.5600, Y 71.0785, Z -2.1667, A 0.000, B 0.000, C 0.000 }
gfCNCPoint1[20059] = {X 353.0406, Y 70.2725, Z -2.1667, A 0.000, B 0.000, C 0.000 }
gfCNCPoint1[20060] = {X 352.5573, Y 69.4443, Z -2.1667, A 0.000, B 0.000, C 0.000 }
gfCNCPoint1[20061] = {X 351.9696, Y 68.3059, Z -2.1667, A 0.000, B 0.000, C 0.000 }
gfCNCPoint1[20062] = {X 351.4501, Y 67.1348, Z -2.1667, A 0.000, B 0.000, C 0.000 }
gfCNCPoint1[20063] = {X 350.6291, Y 67.2153, Z -2.1667, A 0.000, B 0.000, C 0.000 }
gfCNCPoint1[20064] = {X 349.8066, Y 67.2788, Z -2.1667, A 0.000, B 0.000, C 0.000 }
gfCNCPoint1[20065] = {X 349.6465, Y 64.8842, Z -2.1667, A 0.000, B 0.000, C 0.000 }
gfCNCPoint1[20066] = {X 348.4627, Y 64.9446, Z -2.1667, A 0.000, B 0.000, C 0.000 }
gfCNCPoint1[20067] = {X 347.2777, Y 64.9677, Z -2.1667, A 0.000, B 0.000, C 0.000 }
gfCNCPoint1[20068] = {X 344.9730, Y 64.9478, Z -2.1667, A 0.000, B 0.000, C 0.000 }
gfCNCPoint1[20069] = {X 342.6737, Y 64.7909, Z -2.1667, A 0.000, B 0.000, C 0.000 }
gfCNCPoint1[20070] = {X 341.9388, Y 66.7260, Z -2.1667, A 0.000, B 0.000, C 0.000 }
gfCNCPoint1[20071] = {X 341.0011, Y 68.5714, Z -2.1667, A 0.000, B 0.000, C 0.000 }
gfCNCPoint1[20072] = {X 339.8713, Y 70.3058, Z -2.1667, A 0.000, B 0.000, C 0.000 }
gfCNCPoint1[20073] = {X 339.8717, Y 75.1896, Z -2.1667, A 0.000, B 0.000, C 0.000 }
gfCNCPoint1[20074] = {X 343.8291, Y 75.3741, Z -2.1667, A 0.000, B 0.000, C 0.000 }
gfCNCPoint1[20075] = {X 347.7906, Y 75.4139, Z -2.1667, A 0.000, B 0.000, C 0.000 }
gfCNCPoint1[20076] = {X 351.8776, Y 75.3782, Z -2.1667, A 0.000, B 0.000, C 0.000 }
gfCNCPoint1[20077] = {X 355.9604, Y 75.1865, Z -2.1667, A 0.000, B 0.000, C 0.000 }
gfCNCPoint1[20078] = {X 355.9600, Y 70.3194, Z -2.1667, A 0.000, B 0.000, C 0.000 }
gfCNCPoint1[20079] = {X 355.0522, Y 68.9618, Z -2.1667, A 0.000, B 0.000, C 0.000 }
gfCNCPoint1[20080] = {X 354.2627, Y 67.5322, Z -2.1667, A 0.000, B 0.000, C 0.000 }
gfCNCPoint1[20081] = {X 353.5969, Y 66.0409, Z -2.1667, A 0.000, B 0.000, C 0.000 }
gfCNCPoint1[20082] = {X 353.0597, Y 64.4986, Z -2.1667, A 0.000, B 0.000, C 0.000 }
gfCNCPoint1[20083] = {X 351.3575, Y 64.7304, Z -2.1667, A 0.000, B 0.000, C 0.000 }
gfCNCPoint1[20084] = {X 349.6465, Y 64.8842, Z -2.1667, A 0.000, B 0.000, C 0.000 }
gfCNCPoint1[20085] = {X 349.4863, Y 62.4895, Z -2.1667, A 0.000, B 0.000, C 0.000 }
gfCNCPoint1[20086] = {X 348.3677, Y 62.5465, Z -2.1667, A 0.000, B 0.000, C 0.000 }
gfCNCPoint1[20087] = {X 347.2479, Y 62.5678, Z -2.1667, A 0.000, B 0.000, C 0.000 }
gfCNCPoint1[20088] = {X 345.1177, Y 62.5515, Z -2.1667, A 0.000, B 0.000, C 0.000 }
gfCNCPoint1[20089] = {X 342.9921, Y 62.4105, Z -2.1667, A 0.000, B 0.000, C 0.000 }
gfCNCPoint1[20090] = {X 340.8784, Y 62.1453, Z -2.1667, A 0.000, B 0.000, C 0.000 }
gfCNCPoint1[20091] = {X 340.4884, Y 63.7334, Z -2.1667, A 0.000, B 0.000, C 0.000 }
gfCNCPoint1[20092] = {X 339.9470, Y 65.2763, Z -2.1667, A 0.000, B 0.000, C 0.000 }
gfCNCPoint1[20093] = {X 339.2592, Y 66.7598, Z -2.1667, A 0.000, B 0.000, C 0.000 }
gfCNCPoint1[20094] = {X 338.4313, Y 68.1700, Z -2.1667, A 0.000, B 0.000, C 0.000 }
gfCNCPoint1[20095] = {X 337.4713, Y 69.4937, Z -2.1667, A 0.000, B 0.000, C 0.000 }
gfCNCPoint1[20096] = {X 337.4718, Y 77.4159, Z -2.1667, A 0.000, B 0.000, C 0.000 }
gfCNCPoint1[20097] = {X 340.9059, Y 77.6554, Z -2.1667, A 0.000, B 0.000, C 0.000 }
gfCNCPoint1[20098] = {X 344.3457, Y 77.7882, Z -2.1667, A 0.000, B 0.000, C 0.000 }
gfCNCPoint1[20099] = {X 347.7880, Y 77.8139, Z -2.1667, A 0.000, B 0.000, C 0.000 }
gfCNCPoint1[20100] = {X 351.3159, Y 77.7930, Z -2.1667, A 0.000, B 0.000, C 0.000 }
gfCNCPoint1[20101] = {X 354.8413, Y 77.6582, Z -2.1667, A 0.000, B 0.000, C 0.000 }
gfCNCPoint1[20102] = {X 358.3606, Y 77.4098, Z -2.1667, A 0.000, B 0.000, C 0.000 }
gfCNCPoint1[20103] = {X 358.3599, Y 69.5060, Z -2.1667, A 0.000, B 0.000, C 0.000 }
gfCNCPoint1[20104] = {X 357.3487, Y 68.1063, Z -2.1667, A 0.000, B 0.000, C 0.000 }
gfCNCPoint1[20105] = {X 356.4858, Y 66.6107, Z -2.1667, A 0.000, B 0.000, C 0.000 }
gfCNCPoint1[20106] = {X 355.7802, Y 65.0347, Z -2.1667, A 0.000, B 0.000, C 0.000 }
gfCNCPoint1[20107] = {X 355.2394, Y 63.3948, Z -2.1667, A 0.000, B 0.000, C 0.000 }
gfCNCPoint1[20108] = {X 354.8688, Y 61.7083, Z -2.1667, A 0.000, B 0.000, C 0.000 }
gfCNCPoint1[20109] = {X 352.1927, Y 62.2031, Z -2.1667, A 0.000, B 0.000, C 0.000 }
gfCNCPoint1[20110] = {X 349.4863, Y 62.4895, Z -2.1667, A 0.000, B 0.000, C 0.000 }
gfCNCPoint1[20111] = {X 349.3262, Y 60.0949, Z -2.1667, A 0.000, B 0.000, C 0.000 }
gfCNCPoint1[20112] = {X 348.2728, Y 60.1483, Z -2.1667, A 0.000, B 0.000, C 0.000 }
gfCNCPoint1[20113] = {X 347.2182, Y 60.1679, Z -2.1667, A 0.000, B 0.000, C 0.000 }
gfCNCPoint1[20114] = {X 344.3864, Y 60.1129, Z -2.1667, A 0.000, B 0.000, C 0.000 }
gfCNCPoint1[20115] = {X 341.5690, Y 59.8222, Z -2.1667, A 0.000, B 0.000, C 0.000 }
gfCNCPoint1[20116] = {X 338.7856, Y 59.2978, Z -2.1667, A 0.000, B 0.000, C 0.000 }
gfCNCPoint1[20117] = {X 338.6398, Y 60.9973, Z -2.1667, A 0.000, B 0.000, C 0.000 }
gfCNCPoint1[20118] = {X 338.2958, Y 62.6679, Z -2.1667, A 0.000, B 0.000, C 0.000 }
gfCNCPoint1[20119] = {X 337.7582, Y 64.2867, Z -2.1667, A 0.000, B 0.000, C 0.000 }
gfCNCPoint1[20120] = {X 337.0346, Y 65.8312, Z -2.1667, A 0.000, B 0.000, C 0.000 }
gfCNCPoint1[20121] = {X 336.1347, Y 67.2803, Z -2.1667, A 0.000, B 0.000, C 0.000 }
gfCNCPoint1[20122] = {X 335.0712, Y 68.6138, Z -2.1667, A 0.000, B 0.000, C 0.000 }
gfCNCPoint1[20123] = {X 335.0720, Y 79.5889, Z -2.1667, A 0.000, B 0.000, C 0.000 }
gfCNCPoint1[20124] = {X 335.6613, Y 79.6576, Z -2.1667, A 0.000, B 0.000, C 0.000 }
gfCNCPoint1[20125] = {X 336.2518, Y 79.7158, Z -2.1667, A 0.000, B 0.000, C 0.000 }
gfCNCPoint1[20126] = {X 340.0899, Y 80.0127, Z -2.1667, A 0.000, B 0.000, C 0.000 }
gfCNCPoint1[20127] = {X 343.9360, Y 80.1788, Z -2.1667, A 0.000, B 0.000, C 0.000 }
gfCNCPoint1[20128] = {X 347.7854, Y 80.2140, Z -2.1667, A 0.000, B 0.000, C 0.000 }
gfCNCPoint1[20129] = {X 351.8398, Y 80.1810, Z -2.1667, A 0.000, B 0.000, C 0.000 }
gfCNCPoint1[20130] = {X 355.8903, Y 80.0009, Z -2.1667, A 0.000, B 0.000, C 0.000 }
gfCNCPoint1[20131] = {X 359.9315, Y 79.6739, Z -2.1667, A 0.000, B 0.000, C 0.000 }
gfCNCPoint1[20132] = {X 360.3465, Y 79.6323, Z -2.1667, A 0.000, B 0.000, C 0.000 }
gfCNCPoint1[20133] = {X 360.7607, Y 79.5846, Z -2.1667, A 0.000, B 0.000, C 0.000 }
gfCNCPoint1[20134] = {X 360.7598, Y 68.6245, Z -2.1667, A 0.000, B 0.000, C 0.000 }
gfCNCPoint1[20135] = {X 359.7306, Y 67.3422, Z -2.1667, A 0.000, B 0.000, C 0.000 }
gfCNCPoint1[20136] = {X 358.8534, Y 65.9516, Z -2.1667, A 0.000, B 0.000, C 0.000 }
gfCNCPoint1[20137] = {X 358.1395, Y 64.4704, Z -2.1667, A 0.000, B 0.000, C 0.000 }
gfCNCPoint1[20138] = {X 357.5981, Y 62.9178, Z -2.1667, A 0.000, B 0.000, C 0.000 }
gfCNCPoint1[20139] = {X 357.2362, Y 61.3139, Z -2.1667, A 0.000, B 0.000, C 0.000 }
gfCNCPoint1[20140] = {X 357.0916, Y 60.1645, Z -2.1667, A 0.000, B 0.000, C 0.000 }
gfCNCPoint1[20141] = {X 357.0395, Y 59.0073, Z -2.1667, A 0.000, B 0.000, C 0.000 }
gfCNCPoint1[20142] = {X 357.0394, Y 58.6374, Z -2.1667, A 0.000, B 0.000, C 0.000 }
gfCNCPoint1[20143] = {X 355.6983, Y 59.0310, Z -2.1667, A 0.000, B 0.000, C 0.000 }
gfCNCPoint1[20144] = {X 354.3416, Y 59.3670, Z -2.1667, A 0.000, B 0.000, C 0.000 }
gfCNCPoint1[20145] = {X 351.8480, Y 59.8280, Z -2.1667, A 0.000, B 0.000, C 0.000 }
gfCNCPoint1[20146] = {X 349.3262, Y 60.0949, Z -2.1667, A 0.000, B 0.000, C 0.000 }
gfCNCPoint1[20147] = {X 349.1660, Y 57.7002, Z -2.1667, A 0.000, B 0.000, C 0.000 }
gfCNCPoint1[20148] = {X 348.1778, Y 57.7502, Z -2.1667, A 0.000, B 0.000, C 0.000 }
gfCNCPoint1[20149] = {X 347.1885, Y 57.7679, Z -2.1667, A 0.000, B 0.000, C 0.000 }
gfCNCPoint1[20150] = {X 344.5488, Y 57.7184, Z -2.1667, A 0.000, B 0.000, C 0.000 }
gfCNCPoint1[20151] = {X 341.9225, Y 57.4484, Z -2.1667, A 0.000, B 0.000, C 0.000 }
gfCNCPoint1[20152] = {X 339.3279, Y 56.9599, Z -2.1667, A 0.000, B 0.000, C 0.000 }
gfCNCPoint1[20153] = {X 337.7708, Y 56.5567, Z -2.1667, A 0.000, B 0.000, C 0.000 }
gfCNCPoint1[20154] = {X 336.2363, Y 56.0746, Z -2.1667, A 0.000, B 0.000, C 0.000 }
gfCNCPoint1[20155] = {X 336.3520, Y 57.0342, Z -2.1667, A 0.000, B 0.000, C 0.000 }
gfCNCPoint1[20156] = {X 336.3907, Y 58.0000, Z -2.1667, A 0.000, B 0.000, C 0.000 }
gfCNCPoint1[20157] = {X 336.3907, Y 58.9497, Z -2.1667, A 0.000, B 0.000, C 0.000 }
gfCNCPoint1[20158] = {X 336.3894, Y 59.0917, Z -2.1667, A 0.000, B 0.000, C 0.000 }
gfCNCPoint1[20159] = {X 336.3864, Y 59.2336, Z -2.1667, A 0.000, B 0.000, C 0.000 }
gfCNCPoint1[20160] = {X 336.2427, Y 60.7979, Z -2.1667, A 0.000, B 0.000, C 0.000 }
gfCNCPoint1[20161] = {X 335.8978, Y 62.3306, Z -2.1667, A 0.000, B 0.000, C 0.000 }
gfCNCPoint1[20162] = {X 335.3576, Y 63.8057, Z -2.1667, A 0.000, B 0.000, C 0.000 }
gfCNCPoint1[20163] = {X 334.6311, Y 65.1986, Z -2.1667, A 0.000, B 0.000, C 0.000 }
gfCNCPoint1[20164] = {X 333.7306, Y 66.4858, Z -2.1667, A 0.000, B 0.000, C 0.000 }
gfCNCPoint1[20165] = {X 332.6711, Y 67.6457, Z -2.1667, A 0.000, B 0.000, C 0.000 }
gfCNCPoint1[20166] = {X 332.6721, Y 81.6426, Z -2.1667, A 0.000, B 0.000, C 0.000 }
gfCNCPoint1[20167] = {X 334.3494, Y 81.9145, Z -2.1667, A 0.000, B 0.000, C 0.000 }
gfCNCPoint1[20168] = {X 336.0376, Y 82.1063, Z -2.1667, A 0.000, B 0.000, C 0.000 }
gfCNCPoint1[20169] = {X 339.9462, Y 82.4083, Z -2.1667, A 0.000, B 0.000, C 0.000 }
gfCNCPoint1[20170] = {X 343.8628, Y 82.5777, Z -2.1667, A 0.000, B 0.000, C 0.000 }
gfCNCPoint1[20171] = {X 347.7828, Y 82.6141, Z -2.1667, A 0.000, B 0.000, C 0.000 }
gfCNCPoint1[20172] = {X 351.9148, Y 82.5799, Z -2.1667, A 0.000, B 0.000, C 0.000 }
gfCNCPoint1[20173] = {X 356.0428, Y 82.3961, Z -2.1667, A 0.000, B 0.000, C 0.000 }
gfCNCPoint1[20174] = {X 360.1614, Y 82.0629, Z -2.1667, A 0.000, B 0.000, C 0.000 }
gfCNCPoint1[20175] = {X 361.6664, Y 81.8854, Z -2.1667, A 0.000, B 0.000, C 0.000 }
gfCNCPoint1[20176] = {X 363.1609, Y 81.6345, Z -2.1667, A 0.000, B 0.000, C 0.000 }
gfCNCPoint1[20177] = {X 363.1598, Y 67.6544, Z -2.1667, A 0.000, B 0.000, C 0.000 }
gfCNCPoint1[20178] = {X 362.0734, Y 66.4641, Z -2.1667, A 0.000, B 0.000, C 0.000 }
gfCNCPoint1[20179] = {X 361.1551, Y 65.1398, Z -2.1667, A 0.000, B 0.000, C 0.000 }
gfCNCPoint1[20180] = {X 360.4213, Y 63.7050, Z -2.1667, A 0.000, B 0.000, C 0.000 }
gfCNCPoint1[20181] = {X 359.8850, Y 62.1854, Z -2.1667, A 0.000, B 0.000, C 0.000 }
gfCNCPoint1[20182] = {X 359.5558, Y 60.6078, Z -2.1667, A 0.000, B 0.000, C 0.000 }
gfCNCPoint1[20183] = {X 359.4395, Y 59.0005, Z -2.1667, A 0.000, B 0.000, C 0.000 }
gfCNCPoint1[20184] = {X 359.4393, Y 58.0000, Z -2.1667, A 0.000, B 0.000, C 0.000 }
gfCNCPoint1[20185] = {X 359.5345, Y 56.4861, Z -2.1667, A 0.000, B 0.000, C 0.000 }
gfCNCPoint1[20186] = {X 359.8187, Y 54.9962, Z -2.1667, A 0.000, B 0.000, C 0.000 }
gfCNCPoint1[20187] = {X 358.0876, Y 55.7270, Z -2.1667, A 0.000, B 0.000, C 0.000 }
gfCNCPoint1[20188] = {X 356.3147, Y 56.3494, Z -2.1667, A 0.000, B 0.000, C 0.000 }
gfCNCPoint1[20189] = {X 353.9704, Y 56.9900, Z -2.1667, A 0.000, B 0.000, C 0.000 }
gfCNCPoint1[20190] = {X 351.5824, Y 57.4413, Z -2.1667, A 0.000, B 0.000, C 0.000 }
gfCNCPoint1[20191] = {X 349.1660, Y 57.7002, Z -2.1667, A 0.000, B 0.000, C 0.000 }
gfCNCPoint1[20192] = {X 349.0059, Y 55.3056, Z -2.1667, A 0.000, B 0.000, C 0.000 }
gfCNCPoint1[20193] = {X 348.0829, Y 55.3520, Z -2.1667, A 0.000, B 0.000, C 0.000 }
gfCNCPoint1[20194] = {X 347.1589, Y 55.3680, Z -2.1667, A 0.000, B 0.000, C 0.000 }
gfCNCPoint1[20195] = {X 344.5805, Y 55.3157, Z -2.1667, A 0.000, B 0.000, C 0.000 }
gfCNCPoint1[20196] = {X 342.0169, Y 55.0358, Z -2.1667, A 0.000, B 0.000, C 0.000 }
gfCNCPoint1[20197] = {X 339.4880, Y 54.5306, Z -2.1667, A 0.000, B 0.000, C 0.000 }
gfCNCPoint1[20198] = {X 337.0136, Y 53.8040, Z -2.1667, A 0.000, B 0.000, C 0.000 }
gfCNCPoint1[20199] = {X 334.7561, Y 52.9248, Z -2.1667, A 0.000, B 0.000, C 0.000 }
gfCNCPoint1[20200] = {X 332.5794, Y 51.8613, Z -2.1667, A 0.000, B 0.000, C 0.000 }
gfCNCPoint1[20201] = {X 331.5778, Y 51.2711, Z -2.1667, A 0.000, B 0.000, C 0.000 }
gfCNCPoint1[20202] = {X 330.6003, Y 50.6418, Z -2.1667, A 0.000, B 0.000, C 0.000 }
gfCNCPoint1[20203] = {X 331.5700, Y 51.5965, Z -2.1667, A 0.000, B 0.000, C 0.000 }
gfCNCPoint1[20204] = {X 332.3962, Y 52.6777, Z -2.1667, A 0.000, B 0.000, C 0.000 }
gfCNCPoint1[20205] = {X 333.0627, Y 53.8642, Z -2.1667, A 0.000, B 0.000, C 0.000 }
gfCNCPoint1[20206] = {X 333.5562, Y 55.1323, Z -2.1667, A 0.000, B 0.000, C 0.000 }
gfCNCPoint1[20207] = {X 333.8669, Y 56.4572, Z -2.1667, A 0.000, B 0.000, C 0.000 }
gfCNCPoint1[20208] = {X 333.9597, Y 57.2261, Z -2.1667, A 0.000, B 0.000, C 0.000 }
gfCNCPoint1[20209] = {X 333.9907, Y 58.0000, Z -2.1667, A 0.000, B 0.000, C 0.000 }
gfCNCPoint1[20210] = {X 333.9907, Y 58.9452, Z -2.1667, A 0.000, B 0.000, C 0.000 }
gfCNCPoint1[20211] = {X 333.8757, Y 60.4002, Z -2.1667, A 0.000, B 0.000, C 0.000 }
gfCNCPoint1[20212] = {X 333.5442, Y 61.8215, Z -2.1667, A 0.000, B 0.000, C 0.000 }
gfCNCPoint1[20213] = {X 333.0036, Y 63.1771, Z -2.1667, A 0.000, B 0.000, C 0.000 }
gfCNCPoint1[20214] = {X 332.2661, Y 64.4365, Z -2.1667, A 0.000, B 0.000, C 0.000 }
gfCNCPoint1[20215] = {X 331.3484, Y 65.5713, Z -2.1667, A 0.000, B 0.000, C 0.000 }
gfCNCPoint1[20216] = {X 330.2710, Y 66.5559, Z -2.1667, A 0.000, B 0.000, C 0.000 }
gfCNCPoint1[20217] = {X 330.2722, Y 83.2031, Z -2.1667, A 0.000, B 0.000, C 0.000 }
gfCNCPoint1[20218] = {X 330.2760, Y 83.5837, Z -2.1667, A 0.000, B 0.000, C 0.000 }
gfCNCPoint1[20219] = {X 330.3824, Y 83.6090, Z -2.1667, A 0.000, B 0.000, C 0.000 }
gfCNCPoint1[20220] = {X 333.0869, Y 84.1513, Z -2.1667, A 0.000, B 0.000, C 0.000 }
gfCNCPoint1[20221] = {X 335.8235, Y 84.4967, Z -2.1667, A 0.000, B 0.000, C 0.000 }
gfCNCPoint1[20222] = {X 339.8025, Y 84.8040, Z -2.1667, A 0.000, B 0.000, C 0.000 }
gfCNCPoint1[20223] = {X 343.7896, Y 84.9766, Z -2.1667, A 0.000, B 0.000, C 0.000 }
gfCNCPoint1[20224] = {X 347.7803, Y 85.0142, Z -2.1667, A 0.000, B 0.000, C 0.000 }
gfCNCPoint1[20225] = {X 351.9898, Y 84.9787, Z -2.1667, A 0.000, B 0.000, C 0.000 }
gfCNCPoint1[20226] = {X 356.1954, Y 84.7912, Z -2.1667, A 0.000, B 0.000, C 0.000 }
gfCNCPoint1[20227] = {X 360.3914, Y 84.4519, Z -2.1667, A 0.000, B 0.000, C 0.000 }
gfCNCPoint1[20228] = {X 362.9939, Y 84.1050, Z -2.1667, A 0.000, B 0.000, C 0.000 }
gfCNCPoint1[20229] = {X 365.5611, Y 83.5549, Z -2.1667, A 0.000, B 0.000, C 0.000 }
gfCNCPoint1[20230] = {X 365.5597, Y 66.5620, Z -2.1667, A 0.000, B 0.000, C 0.000 }
gfCNCPoint1[20231] = {X 364.4850, Y 65.5840, Z -2.1667, A 0.000, B 0.000, C 0.000 }
gfCNCPoint1[20232] = {X 363.5689, Y 64.4562, Z -2.1667, A 0.000, B 0.000, C 0.000 }
gfCNCPoint1[20233] = {X 362.8319, Y 63.2040, Z -2.1667, A 0.000, B 0.000, C 0.000 }
gfCNCPoint1[20234] = {X 362.2906, Y 61.8555, Z -2.1667, A 0.000, B 0.000, C 0.000 }
gfCNCPoint1[20235] = {X 361.9573, Y 60.4412, Z -2.1667, A 0.000, B 0.000, C 0.000 }
gfCNCPoint1[20236] = {X 361.8395, Y 58.9930, Z -2.1667, A 0.000, B 0.000, C 0.000 }
gfCNCPoint1[20237] = {X 361.8393, Y 58.0000, Z -2.1667, A 0.000, B 0.000, C 0.000 }
gfCNCPoint1[20238] = {X 361.9156, Y 56.7869, Z -2.1667, A 0.000, B 0.000, C 0.000 }
gfCNCPoint1[20239] = {X 362.1433, Y 55.5930, Z -2.1667, A 0.000, B 0.000, C 0.000 }
gfCNCPoint1[20240] = {X 362.5748, Y 54.2989, Z -2.1667, A 0.000, B 0.000, C 0.000 }
gfCNCPoint1[20241] = {X 363.1839, Y 53.0783, Z -2.1667, A 0.000, B 0.000, C 0.000 }
gfCNCPoint1[20242] = {X 363.9585, Y 51.9554, Z -2.1667, A 0.000, B 0.000, C 0.000 }
gfCNCPoint1[20243] = {X 364.8833, Y 50.9526, Z -2.1667, A 0.000, B 0.000, C 0.000 }
gfCNCPoint1[20244] = {X 365.9399, Y 50.0897, Z -2.1667, A 0.000, B 0.000, C 0.000 }
gfCNCPoint1[20245] = {X 367.1072, Y 49.3840, Z -2.1667, A 0.000, B 0.000, C 0.000 }
gfCNCPoint1[20246] = {X 368.3622, Y 48.8493, Z -2.1667, A 0.000, B 0.000, C 0.000 }
gfCNCPoint1[20247] = {X 369.6799, Y 48.4964, Z -2.1667, A 0.000, B 0.000, C 0.000 }
gfCNCPoint1[20248] = {X 371.0341, Y 48.3322, Z -2.1667, A 0.000, B 0.000, C 0.000 }
gfCNCPoint1[20249] = {X 371.2766, Y 48.3230, Z -2.1667, A 0.000, B 0.000, C 0.000 }
gfCNCPoint1[20250] = {X 371.5193, Y 48.3200, Z -2.1667, A 0.000, B 0.000, C 0.000 }
gfCNCPoint1[20251] = {X 388.0597, Y 48.3200, Z -2.1667, A 0.000, B 0.000, C 0.000 }
gfCNCPoint1[20252] = {X 389.4419, Y 48.4192, Z -2.1667, A 0.000, B 0.000, C 0.000 }
gfCNCPoint1[20253] = {X 390.7958, Y 48.7147, Z -2.1667, A 0.000, B 0.000, C 0.000 }
gfCNCPoint1[20254] = {X 392.0936, Y 49.2006, Z -2.1667, A 0.000, B 0.000, C 0.000 }
gfCNCPoint1[20255] = {X 393.3087, Y 49.8667, Z -2.1667, A 0.000, B 0.000, C 0.000 }
gfCNCPoint1[20256] = {X 394.5333, Y 49.1962, Z -2.1667, A 0.000, B 0.000, C 0.000 }
gfCNCPoint1[20257] = {X 395.8416, Y 48.7089, Z -2.1667, A 0.000, B 0.000, C 0.000 }
gfCNCPoint1[20258] = {X 397.1858, Y 48.4177, Z -2.1667, A 0.000, B 0.000, C 0.000 }
gfCNCPoint1[20259] = {X 398.5577, Y 48.3200, Z -2.1667, A 0.000, B 0.000, C 0.000 }
gfCNCPoint1[20260] = {X 398.7346, Y 48.3200, Z -2.1667, A 0.000, B 0.000, C 0.000 }
gfCNCPoint1[20261] = {X 398.1859, Y 47.6069, Z -2.1667, A 0.000, B 0.000, C 0.000 }
gfCNCPoint1[20262] = {X 397.7774, Y 46.8051, Z -2.1667, A 0.000, B 0.000, C 0.000 }
gfCNCPoint1[20263] = {X 397.5230, Y 45.9420, Z -2.1667, A 0.000, B 0.000, C 0.000 }
gfCNCPoint1[20264] = {X 397.4561, Y 45.4921, Z -2.1667, A 0.000, B 0.000, C 0.000 }
gfCNCPoint1[20265] = {X 397.4314, Y 45.0378, Z -2.1667, A 0.000, B 0.000, C 0.000 }
gfCNCPoint1[20266] = {X 397.4316, Y 44.1455, Z -2.1667, A 0.000, B 0.000, C 0.000 }
gfCNCPoint1[20267] = {X 397.5413, Y 43.1779, Z -2.1667, A 0.000, B 0.000, C 0.000 }
gfCNCPoint1[20268] = {X 397.8410, Y 42.2514, Z -2.1667, A 0.000, B 0.000, C 0.000 }
gfCNCPoint1[20269] = {X 398.3186, Y 41.4028, Z -2.1667, A 0.000, B 0.000, C 0.000 }
gfCNCPoint1[20270] = {X 398.9552, Y 40.6660, Z -2.1667, A 0.000, B 0.000, C 0.000 }
gfCNCPoint1[20271] = {X 398.9552, Y 31.8215, Z -2.1667, A 0.000, B 0.000, C 0.000 }
gfCNCPoint1[20272] = {X 396.7496, Y 27.9862, Z -2.1667, A 0.000, B 0.000, C 0.000 }
gfCNCPoint1[20273] = {X 386.3471, Y 33.9685, Z -2.1667, A 0.000, B 0.000, C 0.000 }
gfCNCPoint1[20274] = {X 386.2660, Y 34.3965, Z -2.1667, A 0.000, B 0.000, C 0.000 }
gfCNCPoint1[20275] = {X 386.1812, Y 34.8239, Z -2.1667, A 0.000, B 0.000, C 0.000 }
gfCNCPoint1[20276] = {X 386.0221, Y 35.5735, Z -2.1667, A 0.000, B 0.000, C 0.000 }
gfCNCPoint1[20277] = {X 385.8494, Y 36.3200, Z -2.1667, A 0.000, B 0.000, C 0.000 }
gfCNCPoint1[20278] = {X 386.9552, Y 36.3200, Z -2.1667, A 0.000, B 0.000, C 0.000 }
gfCNCPoint1[20279] = {X 386.9552, Y 35.0259, Z -2.1667, A 0.000, B 0.000, C 0.000 }
gfCNCPoint1[20280] = {X 386.3471, Y 33.9685, Z -2.1667, A 0.000, B 0.000, C 0.000 }
gfCNCPoint1[20281] = {X 388.4276, Y 32.7720, Z -2.1667, A 0.000, B 0.000, C 0.000 }
gfCNCPoint1[20282] = {X 384.7439, Y 26.3664, Z -2.1667, A 0.000, B 0.000, C 0.000 }
gfCNCPoint1[20283] = {X 384.6150, Y 28.7671, Z -2.1667, A 0.000, B 0.000, C 0.000 }
gfCNCPoint1[20284] = {X 384.3625, Y 31.1579, Z -2.1667, A 0.000, B 0.000, C 0.000 }
gfCNCPoint1[20285] = {X 383.9870, Y 33.5325, Z -2.1667, A 0.000, B 0.000, C 0.000 }
gfCNCPoint1[20286] = {X 383.9099, Y 33.9400, Z -2.1667, A 0.000, B 0.000, C 0.000 }
gfCNCPoint1[20287] = {X 383.8291, Y 34.3467, Z -2.1667, A 0.000, B 0.000, C 0.000 }
gfCNCPoint1[20288] = {X 383.6791, Y 35.0536, Z -2.1667, A 0.000, B 0.000, C 0.000 }
gfCNCPoint1[20289] = {X 383.5162, Y 35.7576, Z -2.1667, A 0.000, B 0.000, C 0.000 }
gfCNCPoint1[20290] = {X 383.1264, Y 37.2470, Z -2.1667, A 0.000, B 0.000, C 0.000 }
gfCNCPoint1[20291] = {X 382.6787, Y 38.7200, Z -2.1667, A 0.000, B 0.000, C 0.000 }
gfCNCPoint1[20292] = {X 388.0597, Y 38.7200, Z -2.1667, A 0.000, B 0.000, C 0.000 }
gfCNCPoint1[20293] = {X 388.4821, Y 38.7246, Z -2.1667, A 0.000, B 0.000, C 0.000 }
gfCNCPoint1[20294] = {X 388.9043, Y 38.7385, Z -2.1667, A 0.000, B 0.000, C 0.000 }
gfCNCPoint1[20295] = {X 389.1204, Y 38.2363, Z -2.1667, A 0.000, B 0.000, C 0.000 }
gfCNCPoint1[20296] = {X 389.3552, Y 37.7427, Z -2.1667, A 0.000, B 0.000, C 0.000 }
gfCNCPoint1[20297] = {X 389.3552, Y 34.3850, Z -2.1667, A 0.000, B 0.000, C 0.000 }
gfCNCPoint1[20298] = {X 388.4276, Y 32.7720, Z -2.1667, A 0.000, B 0.000, C 0.000 }
gfCNCPoint1[20299] = {X 390.5081, Y 31.5756, Z -2.1667, A 0.000, B 0.000, C 0.000 }
gfCNCPoint1[20300] = {X 386.5937, Y 24.7689, Z -2.1667, A 0.000, B 0.000, C 0.000 }
gfCNCPoint1[20301] = {X 386.0557, Y 23.8515, Z -2.1667, A 0.000, B 0.000, C 0.000 }
gfCNCPoint1[20302] = {X 385.5019, Y 22.9434, Z -2.1667, A 0.000, B 0.000, C 0.000 }
gfCNCPoint1[20303] = {X 384.4720, Y 22.1532, Z -2.1667, A 0.000, B 0.000, C 0.000 }
gfCNCPoint1[20304] = {X 383.5328, Y 21.2571, Z -2.1667, A 0.000, B 0.000, C 0.000 }
gfCNCPoint1[20305] = {X 382.6952, Y 20.2653, Z -2.1667, A 0.000, B 0.000, C 0.000 }
gfCNCPoint1[20306] = {X 381.9689, Y 19.1894, Z -2.1667, A 0.000, B 0.000, C 0.000 }
gfCNCPoint1[20307] = {X 382.2216, Y 21.5516, Z -2.1667, A 0.000, B 0.000, C 0.000 }
gfCNCPoint1[20308] = {X 382.3471, Y 23.9240, Z -2.1667, A 0.000, B 0.000, C 0.000 }
gfCNCPoint1[20309] = {X 382.3448, Y 26.2996, Z -2.1667, A 0.000, B 0.000, C 0.000 }
gfCNCPoint1[20310] = {X 382.2010, Y 28.8382, Z -2.1667, A 0.000, B 0.000, C 0.000 }
gfCNCPoint1[20311] = {X 381.9114, Y 31.3642, Z -2.1667, A 0.000, B 0.000, C 0.000 }
gfCNCPoint1[20312] = {X 381.4770, Y 33.8694, Z -2.1667, A 0.000, B 0.000, C 0.000 }
gfCNCPoint1[20313] = {X 380.9956, Y 35.9390, Z -2.1667, A 0.000, B 0.000, C 0.000 }
gfCNCPoint1[20314] = {X 380.3965, Y 37.9775, Z -2.1667, A 0.000, B 0.000, C 0.000 }
gfCNCPoint1[20315] = {X 379.8410, Y 39.5622, Z -2.1667, A 0.000, B 0.000, C 0.000 }
gfCNCPoint1[20316] = {X 379.2143, Y 41.1200, Z -2.1667, A 0.000, B 0.000, C 0.000 }
gfCNCPoint1[20317] = {X 388.0597, Y 41.1200, Z -2.1667, A 0.000, B 0.000, C 0.000 }
gfCNCPoint1[20318] = {X 389.3256, Y 41.1675, Z -2.1667, A 0.000, B 0.000, C 0.000 }
gfCNCPoint1[20319] = {X 390.5843, Y 41.3099, Z -2.1667, A 0.000, B 0.000, C 0.000 }
gfCNCPoint1[20320] = {X 391.0709, Y 39.7838, Z -2.1667, A 0.000, B 0.000, C 0.000 }
gfCNCPoint1[20321] = {X 391.7552, Y 38.3355, Z -2.1667, A 0.000, B 0.000, C 0.000 }
gfCNCPoint1[20322] = {X 391.7552, Y 33.7442, Z -2.1667, A 0.000, B 0.000, C 0.000 }
gfCNCPoint1[20323] = {X 390.5081, Y 31.5756, Z -2.1667, A 0.000, B 0.000, C 0.000 }
gfCNCPoint1[20324] = {X 392.5886, Y 30.3791, Z -2.1667, A 0.000, B 0.000, C 0.000 }
gfCNCPoint1[20325] = {X 388.6743, Y 23.5724, Z -2.1667, A 0.000, B 0.000, C 0.000 }
gfCNCPoint1[20326] = {X 387.9769, Y 22.3891, Z -2.1667, A 0.000, B 0.000, C 0.000 }
gfCNCPoint1[20327] = {X 387.2545, Y 21.2209, Z -2.1667, A 0.000, B 0.000, C 0.000 }
gfCNCPoint1[20328] = {X 386.3064, Y 20.5558, Z -2.1667, A 0.000, B 0.000, C 0.000 }
gfCNCPoint1[20329] = {X 385.4445, Y 19.7822, Z -2.1667, A 0.000, B 0.000, C 0.000 }
gfCNCPoint1[20330] = {X 384.6812, Y 18.9113, Z -2.1667, A 0.000, B 0.000, C 0.000 }
gfCNCPoint1[20331] = {X 384.0273, Y 17.9554, Z -2.1667, A 0.000, B 0.000, C 0.000 }
gfCNCPoint1[20332] = {X 383.4394, Y 16.8078, Z -2.1667, A 0.000, B 0.000, C 0.000 }
gfCNCPoint1[20333] = {X 383.0093, Y 15.5922, Z -2.1667, A 0.000, B 0.000, C 0.000 }
gfCNCPoint1[20334] = {X 382.7445, Y 14.3302, Z -2.1667, A 0.000, B 0.000, C 0.000 }
gfCNCPoint1[20335] = {X 382.6498, Y 13.0443, Z -2.1667, A 0.000, B 0.000, C 0.000 }
gfCNCPoint1[20336] = {X 382.6496, Y 12.1868, Z -2.1667, A 0.000, B 0.000, C 0.000 }
gfCNCPoint1[20337] = {X 382.6507, Y 12.0459, Z -2.1667, A 0.000, B 0.000, C 0.000 }
gfCNCPoint1[20338] = {X 382.6537, Y 11.9051, Z -2.1667, A 0.000, B 0.000, C 0.000 }
gfCNCPoint1[20339] = {X 377.7922, Y 11.9051, Z -2.1667, A 0.000, B 0.000, C 0.000 }
gfCNCPoint1[20340] = {X 378.4194, Y 13.8576, Z -2.1667, A 0.000, B 0.000, C 0.000 }
gfCNCPoint1[20341] = {X 378.9307, Y 15.8436, Z -2.1667, A 0.000, B 0.000, C 0.000 }
gfCNCPoint1[20342] = {X 379.3013, Y 17.6689, Z -2.1667, A 0.000, B 0.000, C 0.000 }
gfCNCPoint1[20343] = {X 379.5902, Y 19.5088, Z -2.1667, A 0.000, B 0.000, C 0.000 }
gfCNCPoint1[20344] = {X 379.8690, Y 22.2855, Z -2.1667, A 0.000, B 0.000, C 0.000 }
gfCNCPoint1[20345] = {X 379.9619, Y 25.0747, Z -2.1667, A 0.000, B 0.000, C 0.000 }
gfCNCPoint1[20346] = {X 379.8684, Y 27.8638, Z -2.1667, A 0.000, B 0.000, C 0.000 }
gfCNCPoint1[20347] = {X 379.5890, Y 30.6404, Z -2.1667, A 0.000, B 0.000, C 0.000 }
gfCNCPoint1[20348] = {X 379.1250, Y 33.3922, Z -2.1667, A 0.000, B 0.000, C 0.000 }
gfCNCPoint1[20349] = {X 378.5748, Y 35.6994, Z -2.1667, A 0.000, B 0.000, C 0.000 }
gfCNCPoint1[20350] = {X 377.8682, Y 37.9635, Z -2.1667, A 0.000, B 0.000, C 0.000 }
gfCNCPoint1[20351] = {X 377.0085, Y 40.1741, Z -2.1667, A 0.000, B 0.000, C 0.000 }
gfCNCPoint1[20352] = {X 376.2269, Y 41.8693, Z -2.1667, A 0.000, B 0.000, C 0.000 }
gfCNCPoint1[20353] = {X 375.3551, Y 43.5200, Z -2.1667, A 0.000, B 0.000, C 0.000 }
gfCNCPoint1[20354] = {X 388.0597, Y 43.5200, Z -2.1667, A 0.000, B 0.000, C 0.000 }
gfCNCPoint1[20355] = {X 389.6072, Y 43.6029, Z -2.1667, A 0.000, B 0.000, C 0.000 }
gfCNCPoint1[20356] = {X 391.1370, Y 43.8508, Z -2.1667, A 0.000, B 0.000, C 0.000 }
gfCNCPoint1[20357] = {X 392.6316, Y 44.2607, Z -2.1667, A 0.000, B 0.000, C 0.000 }
gfCNCPoint1[20358] = {X 392.7236, Y 42.8756, Z -2.1667, A 0.000, B 0.000, C 0.000 }
gfCNCPoint1[20359] = {X 393.0129, Y 41.5179, Z -2.1667, A 0.000, B 0.000, C 0.000 }
gfCNCPoint1[20360] = {X 393.4934, Y 40.2155, Z -2.1667, A 0.000, B 0.000, C 0.000 }
gfCNCPoint1[20361] = {X 394.1552, Y 38.9952, Z -2.1667, A 0.000, B 0.000, C 0.000 }
gfCNCPoint1[20362] = {X 394.1552, Y 33.1033, Z -2.1667, A 0.000, B 0.000, C 0.000 }
gfCNCPoint1[20363] = {X 392.5886, Y 30.3791, Z -2.1667, A 0.000, B 0.000, C 0.000 }
gfCNCPoint1[20364] = {X 394.6691, Y 29.1827, Z -2.1667, A 0.000, B 0.000, C 0.000 }
gfCNCPoint1[20365] = {X 390.7548, Y 22.3760, Z -2.1667, A 0.000, B 0.000, C 0.000 }
gfCNCPoint1[20366] = {X 389.9719, Y 21.0503, Z -2.1667, A 0.000, B 0.000, C 0.000 }
gfCNCPoint1[20367] = {X 389.1588, Y 19.7429, Z -2.1667, A 0.000, B 0.000, C 0.000 }
gfCNCPoint1[20368] = {X 389.0402, Y 19.5699, Z -2.1667, A 0.000, B 0.000, C 0.000 }
gfCNCPoint1[20369] = {X 388.9103, Y 19.4050, Z -2.1667, A 0.000, B 0.000, C 0.000 }
gfCNCPoint1[20370] = {X 387.8205, Y 18.6935, Z -2.1667, A 0.000, B 0.000, C 0.000 }
gfCNCPoint1[20371] = {X 386.8749, Y 17.7993, Z -2.1667, A 0.000, B 0.000, C 0.000 }
gfCNCPoint1[20372] = {X 386.1036, Y 16.7510, Z -2.1667, A 0.000, B 0.000, C 0.000 }
gfCNCPoint1[20373] = {X 385.5313, Y 15.5821, Z -2.1667, A 0.000, B 0.000, C 0.000 }
gfCNCPoint1[20374] = {X 385.1763, Y 14.3300, Z -2.1667, A 0.000, B 0.000, C 0.000 }
gfCNCPoint1[20375] = {X 385.0498, Y 13.0347, Z -2.1667, A 0.000, B 0.000, C 0.000 }
gfCNCPoint1[20376] = {X 385.0496, Y 12.1868, Z -2.1667, A 0.000, B 0.000, C 0.000 }
gfCNCPoint1[20377] = {X 385.0504, Y 12.0809, Z -2.1667, A 0.000, B 0.000, C 0.000 }
gfCNCPoint1[20378] = {X 385.0527, Y 11.9749, Z -2.1667, A 0.000, B 0.000, C 0.000 }
gfCNCPoint1[20379] = {X 385.1994, Y 10.7178, Z -2.1667, A 0.000, B 0.000, C 0.000 }
gfCNCPoint1[20380] = {X 385.5616, Y 9.5051, Z -2.1667, A 0.000, B 0.000, C 0.000 }
gfCNCPoint1[20381] = {X 374.2005, Y 9.5051, Z -2.1667, A 0.000, B 0.000, C 0.000 }
gfCNCPoint1[20382] = {X 374.9078, Y 11.0878, Z -2.1667, A 0.000, B 0.000, C 0.000 }
gfCNCPoint1[20383] = {X 375.5297, Y 12.7059, Z -2.1667, A 0.000, B 0.000, C 0.000 }
gfCNCPoint1[20384] = {X 376.1138, Y 14.5241, Z -2.1667, A 0.000, B 0.000, C 0.000 }
gfCNCPoint1[20385] = {X 376.5899, Y 16.3735, Z -2.1667, A 0.000, B 0.000, C 0.000 }
gfCNCPoint1[20386] = {X 377.1072, Y 19.1021, Z -2.1667, A 0.000, B 0.000, C 0.000 }
gfCNCPoint1[20387] = {X 377.4309, Y 21.8603, Z -2.1667, A 0.000, B 0.000, C 0.000 }
gfCNCPoint1[20388] = {X 377.5595, Y 24.6345, Z -2.1667, A 0.000, B 0.000, C 0.000 }
gfCNCPoint1[20389] = {X 377.4923, Y 27.4109, Z -2.1667, A 0.000, B 0.000, C 0.000 }
gfCNCPoint1[20390] = {X 377.2297, Y 30.1756, Z -2.1667, A 0.000, B 0.000, C 0.000 }
gfCNCPoint1[20391] = {X 376.7729, Y 32.9150, Z -2.1667, A 0.000, B 0.000, C 0.000 }
gfCNCPoint1[20392] = {X 376.1753, Y 35.3678, Z -2.1667, A 0.000, B 0.000, C 0.000 }
gfCNCPoint1[20393] = {X 375.3879, Y 37.7663, Z -2.1667, A 0.000, B 0.000, C 0.000 }
gfCNCPoint1[20394] = {X 374.4154, Y 40.0960, Z -2.1667, A 0.000, B 0.000, C 0.000 }
gfCNCPoint1[20395] = {X 373.2638, Y 42.3425, Z -2.1667, A 0.000, B 0.000, C 0.000 }
gfCNCPoint1[20396] = {X 372.1859, Y 44.1205, Z -2.1667, A 0.000, B 0.000, C 0.000 }
gfCNCPoint1[20397] = {X 370.9957, Y 45.8255, Z -2.1667, A 0.000, B 0.000, C 0.000 }
gfCNCPoint1[20398] = {X 370.9139, Y 45.9352, Z -2.1667, A 0.000, B 0.000, C 0.000 }
gfCNCPoint1[20399] = {X 371.2165, Y 45.9238, Z -2.1667, A 0.000, B 0.000, C 0.000 }
gfCNCPoint1[20400] = {X 371.5193, Y 45.9200, Z -2.1667, A 0.000, B 0.000, C 0.000 }
gfCNCPoint1[20401] = {X 388.0597, Y 45.9200, Z -2.1667, A 0.000, B 0.000, C 0.000 }
gfCNCPoint1[20402] = {X 389.4143, Y 45.9962, Z -2.1667, A 0.000, B 0.000, C 0.000 }
gfCNCPoint1[20403] = {X 390.7519, Y 46.2238, Z -2.1667, A 0.000, B 0.000, C 0.000 }
gfCNCPoint1[20404] = {X 392.0555, Y 46.6000, Z -2.1667, A 0.000, B 0.000, C 0.000 }
gfCNCPoint1[20405] = {X 393.3087, Y 47.1200, Z -2.1667, A 0.000, B 0.000, C 0.000 }
gfCNCPoint1[20406] = {X 394.2237, Y 46.7243, Z -2.1667, A 0.000, B 0.000, C 0.000 }
gfCNCPoint1[20407] = {X 395.1681, Y 46.4053, Z -2.1667, A 0.000, B 0.000, C 0.000 }
gfCNCPoint1[20408] = {X 395.0678, Y 45.7292, Z -2.1667, A 0.000, B 0.000, C 0.000 }
gfCNCPoint1[20409] = {X 395.0314, Y 45.0468, Z -2.1667, A 0.000, B 0.000, C 0.000 }
gfCNCPoint1[20410] = {X 395.0316, Y 44.1296, Z -2.1667, A 0.000, B 0.000, C 0.000 }
gfCNCPoint1[20411] = {X 395.1397, Y 42.9564, Z -2.1667, A 0.000, B 0.000, C 0.000 }
gfCNCPoint1[20412] = {X 395.4356, Y 41.8161, Z -2.1667, A 0.000, B 0.000, C 0.000 }
gfCNCPoint1[20413] = {X 395.9116, Y 40.7384, Z -2.1667, A 0.000, B 0.000, C 0.000 }
gfCNCPoint1[20414] = {X 396.5552, Y 39.7516, Z -2.1667, A 0.000, B 0.000, C 0.000 }
gfCNCPoint1[20415] = {X 396.5552, Y 32.4624, Z -2.1667, A 0.000, B 0.000, C 0.000 }
gfCNCPoint1[20416] = {X 394.6691, Y 29.1827, Z -2.1667, A 0.000, B 0.000, C 0.000 }
gfCNCPoint1[20417] = {X 396.7496, Y 27.9862, Z -2.1667, A 0.000, B 0.000, C 0.000 }
gfCNCPoint1[20418] = {X 392.8353, Y 21.1795, Z -2.1667, A 0.000, B 0.000, C 0.000 }
gfCNCPoint1[20419] = {X 392.0244, Y 19.8063, Z -2.1667, A 0.000, B 0.000, C 0.000 }
gfCNCPoint1[20420] = {X 391.1821, Y 18.4520, Z -2.1667, A 0.000, B 0.000, C 0.000 }
gfCNCPoint1[20421] = {X 390.7983, Y 17.9220, Z -2.1667, A 0.000, B 0.000, C 0.000 }
gfCNCPoint1[20422] = {X 390.3550, Y 17.4407, Z -2.1667, A 0.000, B 0.000, C 0.000 }
gfCNCPoint1[20423] = {X 389.5444, Y 16.9851, Z -2.1667, A 0.000, B 0.000, C 0.000 }
gfCNCPoint1[20424] = {X 388.8349, Y 16.3841, Z -2.1667, A 0.000, B 0.000, C 0.000 }
gfCNCPoint1[20425] = {X 388.2523, Y 15.6595, Z -2.1667, A 0.000, B 0.000, C 0.000 }
gfCNCPoint1[20426] = {X 387.8178, Y 14.8375, Z -2.1667, A 0.000, B 0.000, C 0.000 }
